C03650=1232.776,265.965,-62.554,-176.669,6.395,148.177
C03651=1232.781,265.716,-62.527,-176.671,6.393,148.177
C03652=1232.785,265.468,-62.499,-176.673,6.391,148.177
C03653=1232.790,265.219,-62.472,-176.676,6.389,148.178
C03654=1232.794,264.971,-62.445,-176.679,6.387,148.178
C03655=1232.799,264.722,-62.418,-176.681,6.385,148.178
C03656=1232.803,264.474,-62.390,-176.683,6.383,148.178
C03657=1232.807,264.225,-62.363,-176.686,6.381,148.179
C03658=1232.813,263.953,-62.332,-176.689,6.378,148.179
C03659=1232.817,263.680,-62.303,-176.691,6.376,148.179
C03660=1232.822,263.407,-62.274,-176.694,6.374,148.179
C03661=1232.827,263.135,-62.243,-176.697,6.371,148.180
C03662=1232.832,262.886,-62.216,-176.700,6.370,148.180
C03663=1232.836,262.638,-62.190,-176.702,6.367,148.180
C03664=1232.839,262.390,-62.162,-176.704,6.365,148.180
C03665=1232.844,262.141,-62.135,-176.707,6.364,148.181
C03666=1232.849,261.893,-62.108,-176.709,6.361,148.181
C03667=1232.853,261.644,-62.080,-176.712,6.359,148.181
C03668=1232.858,261.396,-62.053,-176.714,6.358,148.181
C03669=1232.863,261.147,-62.026,-176.716,6.355,148.181
C03670=1232.866,260.898,-62.000,-176.719,6.353,148.182
C03671=1232.871,260.650,-61.972,-176.721,6.352,148.182
C03672=1232.875,260.401,-61.945,-176.724,6.350,148.182
C03673=1232.880,260.153,-61.918,-176.726,6.347,148.182
C03674=1232.885,259.904,-61.891,-176.729,6.346,148.183
C03675=1232.889,259.656,-61.865,-176.731,6.344,148.183
C03676=1232.893,259.408,-61.838,-176.734,6.341,148.183
C03677=1232.898,259.159,-61.811,-176.736,6.340,148.183
C03678=1232.903,258.911,-61.784,-176.739,6.338,148.184
C03679=1232.907,258.661,-61.756,-176.741,6.335,148.184
C03680=1232.911,258.413,-61.730,-176.743,6.334,148.184
C03681=1232.915,258.165,-61.703,-176.746,6.332,148.184
C03682=1232.920,257.916,-61.676,-176.749,6.330,148.185
C03683=1232.924,257.668,-61.649,-176.751,6.328,148.185
C03684=1232.928,257.420,-61.622,-176.753,6.326,148.185
C03685=1232.933,257.171,-61.595,-176.756,6.324,148.185
C03686=1232.938,256.923,-61.568,-176.759,6.322,148.186
C03687=1232.942,256.674,-61.541,-176.761,6.320,148.186
C03688=1232.946,256.426,-61.514,-176.763,6.318,148.186
C03689=1232.951,256.177,-61.488,-176.766,6.316,148.186
C03690=1232.955,255.929,-61.462,-176.768,6.314,148.186
C03691=1232.960,255.680,-61.435,-176.771,6.312,148.187
C03692=1232.965,255.432,-61.407,-176.773,6.310,148.187
C03693=1232.968,255.183,-61.381,-176.776,6.308,148.187
C03694=1232.973,254.935,-61.354,-176.778,6.306,148.187
C03695=1232.978,254.686,-61.328,-176.781,6.304,148.188
C03696=1232.981,254.437,-61.301,-176.783,6.302,148.188
C03697=1232.986,254.188,-61.274,-176.786,6.300,148.188
C03698=1232.991,253.940,-61.247,-176.788,6.298,148.188
C03699=1232.995,253.691,-61.221,-176.791,6.296,148.189
C03700=1233.000,253.443,-61.194,-176.793,6.294,148.189
C03701=1233.004,253.194,-61.167,-176.796,6.292,148.189
C03702=1233.008,252.946,-61.140,-176.798,6.290,148.190
C03703=1233.013,252.697,-61.114,-176.800,6.288,148.190
C03704=1233.017,252.449,-61.088,-176.803,6.286,148.190
C03705=1233.022,252.200,-61.060,-176.806,6.284,148.190
C03706=1233.026,251.951,-61.035,-176.808,6.282,148.191
C03707=1233.031,251.704,-61.008,-176.810,6.280,148.191
C03708=1233.035,251.455,-60.982,-176.813,6.278,148.191
C03709=1233.040,251.206,-60.955,-176.816,6.276,148.191
C03710=1233.044,250.958,-60.929,-176.818,6.275,148.192
C03711=1233.049,250.710,-60.902,-176.821,6.273,148.192
C03712=1233.054,250.460,-60.875,-176.823,6.270,148.192
C03713=1233.058,250.212,-60.849,-176.826,6.269,148.192
C03714=1233.062,249.963,-60.823,-176.828,6.267,148.193
C03715=1233.066,249.715,-60.796,-176.831,6.265,148.193
C03716=1233.071,249.466,-60.769,-176.833,6.263,148.193
C03717=1233.075,249.218,-60.743,-176.835,6.261,148.193
C03718=1233.080,248.969,-60.716,-176.838,6.259,148.194
C03719=1233.084,248.720,-60.690,-176.841,6.257,148.194
C03720=1233.088,248.472,-60.664,-176.843,6.255,148.194
C03721=1233.093,248.223,-60.638,-176.846,6.253,148.194
C03722=1233.097,247.975,-60.611,-176.848,6.252,148.195
C03723=1233.103,247.726,-60.585,-176.850,6.250,148.195
C03724=1233.106,247.478,-60.559,-176.853,6.248,148.195
C03725=1233.111,247.229,-60.532,-176.855,6.246,148.196
C03726=1233.115,246.981,-60.506,-176.858,6.244,148.196
C03727=1233.120,246.732,-60.480,-176.860,6.242,148.196
C03728=1233.124,246.484,-60.453,-176.863,6.240,148.196
C03729=1233.128,246.235,-60.427,-176.865,6.238,148.197
C03730=1233.133,245.986,-60.401,-176.868,6.236,148.197
C03731=1233.137,245.738,-60.375,-176.871,6.234,148.197
C03732=1233.142,245.489,-60.349,-176.873,6.233,148.197
C03733=1233.147,245.241,-60.322,-176.875,6.230,148.198
C03734=1233.151,244.992,-60.296,-176.878,6.229,148.198
C03735=1233.156,244.743,-60.270,-176.880,6.227,148.198
C03736=1233.160,244.495,-60.243,-176.883,6.225,148.198
C03737=1233.164,244.246,-60.218,-176.886,6.223,148.199
C03738=1233.169,243.997,-60.191,-176.888,6.221,148.199
C03739=1233.174,243.749,-60.165,-176.890,6.220,148.199
C03740=1233.178,243.501,-60.140,-176.892,6.218,148.200
C03741=1233.183,243.252,-60.113,-176.895,6.216,148.200
C03742=1233.187,243.003,-60.087,-176.898,6.214,148.200
C03743=1233.191,242.755,-60.061,-176.900,6.212,148.200
C03744=1233.196,242.506,-60.036,-176.903,6.210,148.201
C03745=1233.201,242.257,-60.009,-176.906,6.208,148.201
C03746=1233.205,242.009,-59.983,-176.908,6.206,148.201
C03747=1233.209,241.760,-59.957,-176.910,6.204,148.201
C03748=1233.214,241.511,-59.931,-176.913,6.202,148.202
C03749=1233.219,241.263,-59.905,-176.915,6.200,148.202
C03750=1233.223,241.014,-59.880,-176.918,6.199,148.202
C03751=1233.227,240.766,-59.853,-176.921,6.197,148.203
C03752=1233.232,240.517,-59.827,-176.923,6.196,148.203
C03753=1233.236,240.268,-59.801,-176.925,6.194,148.203
C03754=1233.241,240.020,-59.776,-176.928,6.192,148.204
C03755=1233.245,239.771,-59.750,-176.930,6.190,148.204
C03756=1233.249,239.522,-59.724,-176.933,6.188,148.204
C03757=1233.254,239.274,-59.697,-176.935,6.186,148.204
C03758=1233.259,239.026,-59.672,-176.938,6.184,148.205
C03759=1233.263,238.777,-59.646,-176.941,6.182,148.205
C03760=1233.267,238.528,-59.620,-176.943,6.180,148.205
C03761=1233.271,238.279,-59.594,-176.946,6.178,148.206
C03762=1233.277,238.008,-59.567,-176.948,6.176,148.206
C03763=1233.282,237.737,-59.537,-176.951,6.175,148.206
C03764=1233.287,237.466,-59.510,-176.954,6.173,148.207
C03765=1233.292,237.194,-59.482,-176.956,6.171,148.207
C03766=1233.296,236.945,-59.456,-176.959,6.169,148.207
C03767=1233.301,236.697,-59.431,-176.961,6.167,148.208
C03768=1233.305,236.448,-59.405,-176.964,6.165,148.208
C03769=1233.309,236.199,-59.379,-176.967,6.163,148.208
C03770=1233.314,235.951,-59.354,-176.969,6.161,148.208
C03771=1233.318,235.702,-59.328,-176.971,6.159,148.209
C03772=1233.323,235.453,-59.302,-176.974,6.158,148.209
C03773=1233.327,235.205,-59.277,-176.976,6.156,148.209
C03774=1233.332,234.956,-59.250,-176.979,6.154,148.210
C03775=1233.337,234.707,-59.225,-176.981,6.153,148.210
C03776=1233.341,234.459,-59.199,-176.984,6.151,148.210
C03777=1233.346,234.210,-59.174,-176.987,6.149,148.211
C03778=1233.350,233.962,-59.148,-176.989,6.147,148.211
C03779=1233.355,233.714,-59.122,-176.992,6.145,148.211
C03780=1233.359,233.464,-59.097,-176.994,6.144,148.212
C03781=1233.363,233.215,-59.072,-176.997,6.142,148.212
C03782=1233.368,232.967,-59.046,-176.999,6.140,148.212
C03783=1233.373,232.718,-59.020,-177.002,6.138,148.213
C03784=1233.377,232.470,-58.995,-177.004,6.136,148.213
C03785=1233.382,232.221,-58.969,-177.007,6.134,148.213
C03786=1233.386,231.972,-58.944,-177.009,6.132,148.213
C03787=1233.390,231.723,-58.919,-177.012,6.130,148.214
C03788=1233.395,231.475,-58.893,-177.014,6.129,148.214
C03789=1233.399,231.226,-58.867,-177.016,6.128,148.214
C03790=1233.404,230.978,-58.842,-177.019,6.126,148.215
C03791=1233.409,230.729,-58.817,-177.022,6.124,148.215
C03792=1233.413,230.480,-58.791,-177.024,6.122,148.215
C03793=1233.418,230.232,-58.766,-177.027,6.120,148.216
C03794=1233.422,229.983,-58.740,-177.030,6.118,148.216
C03795=1233.427,229.734,-58.715,-177.032,6.117,148.216
C03796=1233.431,229.486,-58.690,-177.034,6.115,148.217
C03797=1233.435,229.237,-58.665,-177.037,6.113,148.217
C03798=1233.440,228.988,-58.640,-177.039,6.111,148.217
C03799=1233.444,228.740,-58.614,-177.042,6.110,148.218
C03800=1233.449,228.491,-58.589,-177.045,6.108,148.218
C03801=1233.454,228.242,-58.564,-177.047,6.106,148.218
C03802=1233.458,227.994,-58.538,-177.049,6.105,148.219
C03803=1233.463,227.745,-58.513,-177.052,6.103,148.219
C03804=1233.468,227.496,-58.488,-177.055,6.101,148.219
C03805=1233.471,227.248,-58.463,-177.057,6.099,148.219
C03806=1233.476,226.998,-58.438,-177.060,6.097,148.220
C03807=1233.481,226.750,-58.412,-177.062,6.095,148.220
C03808=1233.485,226.502,-58.387,-177.065,6.094,148.220
C03809=1233.490,226.253,-58.362,-177.067,6.093,148.221
C03810=1233.494,226.004,-58.336,-177.070,6.091,148.221
C03811=1233.499,225.756,-58.312,-177.072,6.089,148.221
C03812=1233.503,225.507,-58.286,-177.075,6.087,148.222
C03813=1233.508,225.258,-58.262,-177.078,6.085,148.222
C03814=1233.512,225.009,-58.236,-177.080,6.083,148.222
C03815=1233.517,224.761,-58.211,-177.082,6.082,148.223
C03816=1233.521,224.512,-58.186,-177.085,6.080,148.223
C03817=1233.526,224.263,-58.161,-177.088,6.078,148.223
C03818=1233.530,224.015,-58.136,-177.090,6.076,148.224
C03819=1233.535,223.766,-58.111,-177.093,6.075,148.224
C03820=1233.539,223.517,-58.086,-177.095,6.073,148.224
C03821=1233.544,223.269,-58.061,-177.097,6.072,148.225
C03822=1233.548,223.020,-58.035,-177.100,6.070,148.225
C03823=1233.553,222.771,-58.011,-177.103,6.068,148.225
C03824=1233.557,222.522,-57.986,-177.105,6.066,148.226
C03825=1233.562,222.274,-57.961,-177.108,6.064,148.226
C03826=1233.567,222.025,-57.936,-177.111,6.062,148.226
C03827=1233.570,221.777,-57.911,-177.113,6.061,148.227
C03828=1233.576,221.528,-57.886,-177.115,6.059,148.227
C03829=1233.580,221.278,-57.861,-177.118,6.058,148.227
C03830=1233.585,221.030,-57.836,-177.121,6.056,148.228
C03831=1233.589,220.781,-57.812,-177.123,6.054,148.228
C03832=1233.594,220.533,-57.787,-177.126,6.052,148.228
C03833=1233.598,220.284,-57.761,-177.128,6.051,148.229
C03834=1233.603,220.035,-57.737,-177.130,6.049,148.229
C03835=1233.608,219.787,-57.712,-177.133,6.047,148.229
C03836=1233.611,219.538,-57.688,-177.136,6.045,148.230
C03837=1233.616,219.289,-57.663,-177.138,6.043,148.230
C03838=1233.621,219.040,-57.638,-177.140,6.042,148.230
C03839=1233.625,218.792,-57.613,-177.143,6.041,148.231
C03840=1233.630,218.543,-57.589,-177.146,6.039,148.231
C03841=1233.635,218.294,-57.563,-177.148,6.037,148.231
C03842=1233.639,218.046,-57.539,-177.151,6.035,148.232
C03843=1233.643,217.796,-57.514,-177.154,6.033,148.232
C03844=1233.648,217.548,-57.490,-177.156,6.032,148.232
C03845=1233.653,217.299,-57.465,-177.159,6.030,148.233
C03846=1233.656,217.051,-57.440,-177.161,6.029,148.233
C03847=1233.662,216.802,-57.415,-177.164,6.027,148.234
C03848=1233.667,216.553,-57.391,-177.167,6.025,148.234
C03849=1233.671,216.304,-57.366,-177.169,6.024,148.234
C03850=1233.676,216.055,-57.342,-177.171,6.022,148.235
C03851=1233.680,215.807,-57.317,-177.174,6.020,148.235
C03852=1233.685,215.557,-57.292,-177.177,6.018,148.235
C03853=1233.689,215.310,-57.268,-177.179,6.016,148.236
C03854=1233.694,215.061,-57.243,-177.181,6.015,148.236
C03855=1233.698,214.812,-57.219,-177.184,6.013,148.236
C03856=1233.703,214.563,-57.194,-177.187,6.012,148.237
C03857=1233.707,214.315,-57.170,-177.189,6.010,148.237
C03858=1233.712,214.065,-57.145,-177.192,6.008,148.238
C03859=1233.716,213.817,-57.121,-177.194,6.007,148.238
C03860=1233.721,213.568,-57.096,-177.197,6.005,148.238
C03861=1233.725,213.319,-57.072,-177.200,6.003,148.239
C03862=1233.730,213.070,-57.047,-177.202,6.002,148.239
C03863=1233.735,212.822,-57.023,-177.204,6.000,148.239
C03864=1233.738,212.573,-56.998,-177.207,5.999,148.240
C03865=1233.743,212.324,-56.974,-177.210,5.997,148.240
C03866=1233.749,212.054,-56.947,-177.212,5.995,148.240
C03867=1233.753,211.783,-56.922,-177.215,5.993,148.241
C03868=1233.758,211.513,-56.895,-177.218,5.991,148.241
C03869=1233.763,211.242,-56.868,-177.221,5.990,148.242
C03870=1233.767,210.994,-56.844,-177.223,5.988,148.242
C03871=1233.773,210.745,-56.819,-177.226,5.986,148.242
C03872=1233.776,210.496,-56.795,-177.228,5.985,148.243
C03873=1233.782,210.247,-56.771,-177.231,5.983,148.243
C03874=1233.786,209.998,-56.747,-177.234,5.981,148.243
C03875=1233.791,209.750,-56.723,-177.236,5.980,148.244
C03876=1233.796,209.501,-56.698,-177.238,5.979,148.244
C03877=1233.799,209.252,-56.673,-177.241,5.977,148.244
C03878=1233.804,209.004,-56.649,-177.244,5.975,148.245
C03879=1233.809,208.755,-56.625,-177.246,5.973,148.245
C03880=1233.814,208.506,-56.601,-177.248,5.972,148.246
C03881=1233.817,208.257,-56.577,-177.251,5.970,148.246
C03882=1233.823,208.008,-56.552,-177.254,5.968,148.246
C03883=1233.827,207.760,-56.528,-177.257,5.967,148.247
C03884=1233.831,207.511,-56.504,-177.259,5.966,148.247
C03885=1233.837,207.262,-56.480,-177.261,5.964,148.247
C03886=1233.841,207.013,-56.456,-177.264,5.962,148.248
C03887=1233.845,206.764,-56.432,-177.267,5.960,148.248
C03888=1233.850,206.515,-56.408,-177.269,5.959,148.248
C03889=1233.855,206.267,-56.384,-177.272,5.957,148.249
C03890=1233.859,206.018,-56.360,-177.274,5.956,148.249
C03891=1233.864,205.770,-56.335,-177.277,5.954,148.250
C03892=1233.868,205.520,-56.312,-177.279,5.953,148.250
C03893=1233.873,205.271,-56.287,-177.282,5.951,148.250
C03894=1233.877,205.023,-56.263,-177.284,5.949,148.251
C03895=1233.882,204.774,-56.240,-177.287,5.947,148.251
C03896=1233.886,204.526,-56.216,-177.290,5.946,148.252
C03897=1233.892,204.277,-56.191,-177.292,5.945,148.252
C03898=1233.896,204.027,-56.167,-177.295,5.943,148.252
C03899=1233.900,203.779,-56.143,-177.297,5.942,148.253
C03900=1233.905,203.530,-56.120,-177.300,5.940,148.253
C03901=1233.909,203.281,-56.096,-177.302,5.938,148.253
C03902=1233.913,203.033,-56.072,-177.305,5.936,148.254
C03903=1233.919,202.783,-56.048,-177.307,5.935,148.254
C03904=1233.923,202.535,-56.024,-177.310,5.933,148.255
C03905=1233.928,202.286,-56.000,-177.313,5.932,148.255
C03906=1233.932,202.037,-55.976,-177.315,5.931,148.255
C03907=1233.937,201.788,-55.952,-177.317,5.929,148.256
C03908=1233.941,201.539,-55.928,-177.320,5.927,148.256
C03909=1233.946,201.290,-55.905,-177.323,5.925,148.257
C03910=1233.951,201.042,-55.880,-177.325,5.924,148.257
C03911=1233.955,200.793,-55.857,-177.328,5.922,148.257
C03912=1233.960,200.544,-55.833,-177.331,5.921,148.258
C03913=1233.965,200.295,-55.809,-177.333,5.920,148.258
C03914=1233.969,200.047,-55.785,-177.335,5.918,148.258
C03915=1233.974,199.798,-55.762,-177.338,5.916,148.259
C03916=1233.978,199.549,-55.738,-177.341,5.914,148.259
C03917=1233.983,199.300,-55.715,-177.343,5.913,148.260
C03918=1233.987,199.052,-55.691,-177.346,5.911,148.260
C03919=1233.991,198.802,-55.667,-177.348,5.910,148.260
C03920=1233.996,198.553,-55.643,-177.350,5.909,148.261
C03921=1234.000,198.305,-55.619,-177.354,5.907,148.261
C03922=1234.005,198.056,-55.596,-177.356,5.905,148.262
C03923=1234.010,197.807,-55.573,-177.358,5.904,148.262
C03924=1234.015,197.558,-55.548,-177.361,5.902,148.262
C03925=1234.020,197.309,-55.525,-177.364,5.900,148.263
C03926=1234.024,197.060,-55.501,-177.366,5.900,148.263
C03927=1234.029,196.811,-55.477,-177.369,5.898,148.264
C03928=1234.033,196.562,-55.454,-177.371,5.896,148.264
C03929=1234.038,196.313,-55.430,-177.373,5.895,148.264
C03930=1234.042,196.065,-55.407,-177.376,5.893,148.265
C03931=1234.046,195.816,-55.384,-177.379,5.891,148.265
C03932=1234.051,195.567,-55.360,-177.381,5.891,148.266
C03933=1234.055,195.319,-55.336,-177.384,5.889,148.266
C03934=1234.060,195.070,-55.313,-177.387,5.887,148.266
C03935=1234.065,194.821,-55.289,-177.389,5.886,148.267
C03936=1234.070,194.572,-55.266,-177.391,5.884,148.267
C03937=1234.074,194.323,-55.242,-177.394,5.882,148.268
C03938=1234.079,194.074,-55.219,-177.396,5.881,148.268
C03939=1234.083,193.825,-55.195,-177.399,5.880,148.268
C03940=1234.088,193.576,-55.172,-177.402,5.878,148.269
C03941=1234.093,193.327,-55.149,-177.404,5.877,148.269
C03942=1234.097,193.078,-55.125,-177.407,5.875,148.270
C03943=1234.102,192.830,-55.102,-177.410,5.873,148.270
C03944=1234.107,192.581,-55.078,-177.412,5.872,148.270
C03945=1234.111,192.333,-55.055,-177.414,5.870,148.271
C03946=1234.116,192.084,-55.032,-177.417,5.869,148.271
C03947=1234.121,191.835,-55.009,-177.420,5.868,148.272
C03948=1234.125,191.586,-54.985,-177.422,5.866,148.272
C03949=1234.130,191.337,-54.962,-177.425,5.864,148.272
C03950=1234.135,191.087,-54.939,-177.427,5.863,148.273
C03951=1234.139,190.839,-54.915,-177.430,5.862,148.273
C03952=1234.143,190.590,-54.892,-177.432,5.861,148.274
C03953=1234.148,190.341,-54.868,-177.435,5.859,148.274
C03954=1234.152,190.092,-54.845,-177.437,5.857,148.274
C03955=1234.158,189.844,-54.822,-177.440,5.856,148.275
C03956=1234.162,189.595,-54.799,-177.443,5.854,148.275
C03957=1234.166,189.346,-54.776,-177.445,5.853,148.276
C03958=1234.171,189.097,-54.753,-177.447,5.852,148.276
C03959=1234.176,188.848,-54.729,-177.450,5.850,148.276
C03960=1234.180,188.599,-54.706,-177.453,5.849,148.277
C03961=1234.185,188.350,-54.683,-177.455,5.847,148.277
C03962=1234.189,188.101,-54.660,-177.458,5.845,148.278
C03963=1234.194,187.852,-54.636,-177.460,5.844,148.278
C03964=1234.199,187.604,-54.613,-177.463,5.843,148.279
C03965=1234.204,187.355,-54.590,-177.466,5.841,148.279
C03966=1234.208,187.106,-54.567,-177.468,5.840,148.279
C03967=1234.213,186.857,-54.545,-177.470,5.838,148.280
C03968=1234.217,186.608,-54.521,-177.473,5.837,148.280
C03969=1234.221,186.359,-54.499,-177.476,5.835,148.281
C03970=1234.227,186.089,-54.473,-177.478,5.834,148.281
C03971=1234.232,185.820,-54.448,-177.481,5.832,148.282
C03972=1234.236,185.550,-54.423,-177.484,5.831,148.282
C03973=1234.242,185.281,-54.398,-177.487,5.830,148.283
C03974=1234.246,185.032,-54.375,-177.489,5.828,148.283
C03975=1234.251,184.782,-54.353,-177.491,5.827,148.283
C03976=1234.256,184.534,-54.330,-177.494,5.825,148.284
C03977=1234.261,184.285,-54.307,-177.497,5.823,148.284
C03978=1234.265,184.036,-54.284,-177.499,5.822,148.285
C03979=1234.269,183.787,-54.260,-177.502,5.820,148.285
C03980=1234.274,183.538,-54.238,-177.504,5.820,148.286
C03981=1234.279,183.290,-54.215,-177.507,5.818,148.286
C03982=1234.284,183.041,-54.192,-177.510,5.816,148.286
C03983=1234.288,182.791,-54.169,-177.512,5.815,148.287
C03984=1234.293,182.542,-54.147,-177.515,5.814,148.287
C03985=1234.298,182.294,-54.124,-177.517,5.813,148.288
C03986=1234.302,182.045,-54.101,-177.520,5.811,148.288
C03987=1234.307,181.796,-54.077,-177.522,5.809,148.288
C03988=1234.312,181.546,-54.055,-177.525,5.808,148.289
C03989=1234.315,181.298,-54.032,-177.528,5.806,148.289
C03990=1234.321,181.049,-54.009,-177.530,5.805,148.290
C03991=1234.325,180.800,-53.987,-177.533,5.804,148.290
C03992=1234.330,180.551,-53.964,-177.535,5.803,148.291
C03993=1234.334,180.303,-53.941,-177.538,5.801,148.291
C03994=1234.339,180.053,-53.919,-177.540,5.799,148.291
C03995=1234.343,179.805,-53.896,-177.543,5.798,148.292
C03996=1234.348,179.556,-53.872,-177.545,5.797,148.292
C03997=1234.353,179.307,-53.851,-177.547,5.795,148.293
C03998=1234.358,179.058,-53.827,-177.551,5.794,148.293
C03999=1234.362,178.809,-53.805,-177.553,5.793,148.294
C04000=1234.367,178.560,-53.782,-177.555,5.791,148.294
C04001=1234.371,178.311,-53.760,-177.558,5.789,148.294
C04002=1234.376,178.062,-53.737,-177.561,5.789,148.295
C04003=1234.380,177.813,-53.714,-177.563,5.787,148.295
C04004=1234.386,177.564,-53.692,-177.565,5.786,148.296
C04005=1234.390,177.315,-53.669,-177.568,5.784,148.296
C04006=1234.395,177.066,-53.647,-177.571,5.783,148.297
C04007=1234.399,176.818,-53.624,-177.573,5.781,148.297
C04008=1234.404,176.568,-53.602,-177.576,5.781,148.298
C04009=1234.408,176.319,-53.579,-177.578,5.779,148.298
C04010=1234.414,176.070,-53.556,-177.580,5.778,148.298
C04011=1234.418,175.822,-53.534,-177.584,5.776,148.299
C04012=1234.422,175.572,-53.512,-177.586,5.774,148.299
C04013=1234.427,175.324,-53.489,-177.588,5.773,148.300
C04014=1234.432,175.075,-53.467,-177.592,5.772,148.300
C04015=1234.436,174.826,-53.443,-177.594,5.771,148.301
C04016=1234.441,174.577,-53.422,-177.596,5.769,148.301
C04017=1234.445,174.328,-53.400,-177.598,5.768,148.301
C04018=1234.450,174.079,-53.376,-177.601,5.767,148.302
C04019=1234.455,173.830,-53.354,-177.604,5.766,148.302
C04020=1234.460,173.581,-53.331,-177.606,5.764,148.303
C04021=1234.465,173.332,-53.309,-177.609,5.763,148.303
C04022=1234.469,173.083,-53.287,-177.611,5.761,148.304
C04023=1234.473,172.834,-53.264,-177.614,5.760,148.304
C04024=1234.478,172.585,-53.242,-177.617,5.759,148.305
C04025=1234.483,172.336,-53.220,-177.619,5.758,148.305
C04026=1234.488,172.088,-53.197,-177.621,5.756,148.305
C04027=1234.492,171.838,-53.175,-177.624,5.755,148.306
C04028=1234.496,171.589,-53.153,-177.627,5.753,148.306
C04029=1234.502,171.341,-53.130,-177.629,5.751,148.307
C04030=1234.506,171.091,-53.108,-177.632,5.751,148.307
C04031=1234.511,170.843,-53.086,-177.635,5.749,148.308
C04032=1234.516,170.593,-53.064,-177.637,5.748,148.308
C04033=1234.520,170.345,-53.041,-177.640,5.746,148.309
C04034=1234.525,170.096,-53.019,-177.642,5.745,148.309
C04035=1234.529,169.846,-52.997,-177.645,5.744,148.310
C04036=1234.535,169.597,-52.975,-177.647,5.743,148.310
C04037=1234.539,169.349,-52.952,-177.650,5.741,148.310
C04038=1234.543,169.100,-52.931,-177.652,5.740,148.311
C04039=1234.548,168.851,-52.909,-177.655,5.739,148.311
C04040=1234.553,168.602,-52.886,-177.657,5.738,148.312
C04041=1234.558,168.352,-52.864,-177.660,5.736,148.312
C04042=1234.562,168.104,-52.842,-177.662,5.735,148.313
C04043=1234.566,167.855,-52.820,-177.665,5.733,148.313
C04044=1234.571,167.606,-52.798,-177.668,5.733,148.314
C04045=1234.576,167.357,-52.775,-177.670,5.731,148.314
C04046=1234.581,167.108,-52.754,-177.672,5.730,148.314
C04047=1234.585,166.859,-52.732,-177.675,5.728,148.315
C04048=1234.590,166.609,-52.710,-177.678,5.727,148.315
C04049=1234.594,166.361,-52.687,-177.680,5.726,148.316
C04050=1234.599,166.112,-52.665,-177.683,5.725,148.316
C04051=1234.604,165.863,-52.643,-177.685,5.724,148.317
C04052=1234.609,165.614,-52.621,-177.688,5.722,148.317
C04053=1234.613,165.365,-52.599,-177.690,5.721,148.318
C04054=1234.618,165.116,-52.578,-177.693,5.719,148.318
C04055=1234.622,164.867,-52.556,-177.695,5.719,148.319
C04056=1234.627,164.618,-52.534,-177.698,5.717,148.319
C04057=1234.632,164.369,-52.511,-177.701,5.716,148.320
C04058=1234.637,164.120,-52.490,-177.703,5.714,148.320
C04059=1234.641,163.871,-52.467,-177.705,5.713,148.320
C04060=1234.646,163.622,-52.446,-177.709,5.712,148.321
C04061=1234.651,163.373,-52.424,-177.711,5.711,148.321
C04062=1234.655,163.124,-52.402,-177.713,5.709,148.322
C04063=1234.660,162.875,-52.380,-177.716,5.708,148.322
C04064=1234.665,162.626,-52.358,-177.718,5.706,148.323
C04065=1234.669,162.377,-52.336,-177.721,5.706,148.323
C04066=1234.674,162.128,-52.315,-177.723,5.705,148.324
C04067=1234.679,161.880,-52.293,-177.726,5.703,148.324
C04068=1234.683,161.630,-52.271,-177.728,5.702,148.325
C04069=1234.688,161.382,-52.249,-177.731,5.700,148.325
C04070=1234.692,161.132,-52.228,-177.734,5.700,148.326
C04071=1234.698,160.883,-52.206,-177.736,5.698,148.326
C04072=1234.703,160.634,-52.184,-177.738,5.697,148.327
C04073=1234.707,160.385,-52.162,-177.742,5.695,148.327
C04074=1234.711,160.116,-52.138,-177.744,5.694,148.328
C04075=1234.717,159.847,-52.115,-177.747,5.693,148.328
C04076=1234.722,159.578,-52.092,-177.750,5.691,148.329
C04077=1234.727,159.309,-52.068,-177.752,5.690,148.329
C04078=1234.731,159.059,-52.047,-177.755,5.689,148.330
C04079=1234.736,158.811,-52.025,-177.757,5.688,148.330
C04080=1234.741,158.562,-52.003,-177.759,5.687,148.330
C04081=1234.745,158.313,-51.981,-177.763,5.685,148.331
C04082=1234.750,158.064,-51.960,-177.765,5.684,148.331
C04083=1234.756,157.815,-51.939,-177.768,5.683,148.332
C04084=1234.760,157.565,-51.917,-177.770,5.682,148.332
C04085=1234.765,157.317,-51.895,-177.773,5.680,148.333
C04086=1234.769,157.067,-51.873,-177.775,5.679,148.333
C04087=1234.774,156.818,-51.852,-177.778,5.678,148.334
C04088=1234.779,156.569,-51.830,-177.780,5.677,148.334
C04089=1234.783,156.320,-51.808,-177.782,5.676,148.335
C04090=1234.787,156.072,-51.787,-177.786,5.674,148.335
C04091=1234.793,155.823,-51.766,-177.788,5.673,148.336
C04092=1234.797,155.573,-51.744,-177.791,5.672,148.336
C04093=1234.802,155.325,-51.723,-177.793,5.671,148.337
C04094=1234.807,155.075,-51.702,-177.795,5.670,148.337
C04095=1234.812,154.827,-51.680,-177.798,5.668,148.338
C04096=1234.816,154.577,-51.658,-177.800,5.667,148.338
C04097=1234.821,154.328,-51.637,-177.803,5.666,148.339
C04098=1234.825,154.080,-51.616,-177.806,5.665,148.339
C04099=1234.830,153.830,-51.594,-177.808,5.664,148.340
C04100=1234.835,153.581,-51.573,-177.811,5.662,148.340
C04101=1234.840,153.332,-51.551,-177.813,5.662,148.341
C04102=1234.844,153.083,-51.530,-177.816,5.660,148.341
C04103=1234.849,152.834,-51.508,-177.818,5.659,148.342
C04104=1234.853,152.585,-51.488,-177.821,5.657,148.342
C04105=1234.858,152.336,-51.466,-177.823,5.656,148.343
C04106=1234.863,152.086,-51.445,-177.826,5.656,148.343
C04107=1234.868,151.838,-51.423,-177.829,5.654,148.344
C04108=1234.873,151.589,-51.401,-177.831,5.653,148.344
C04109=1234.877,151.340,-51.381,-177.833,5.652,148.345
C04110=1234.881,151.091,-51.359,-177.837,5.651,148.345
C04111=1234.887,150.841,-51.338,-177.839,5.650,148.346
C04112=1234.891,150.593,-51.316,-177.841,5.648,148.346
C04113=1234.896,150.344,-51.296,-177.844,5.647,148.347
C04114=1234.900,150.094,-51.275,-177.846,5.646,148.347
C04115=1234.905,149.845,-51.253,-177.849,5.645,148.348
C04116=1234.910,149.596,-51.232,-177.851,5.644,148.348
C04117=1234.915,149.348,-51.211,-177.854,5.642,148.349
C04118=1234.920,149.098,-51.190,-177.857,5.641,148.349
C04119=1234.924,148.849,-51.168,-177.859,5.641,148.350
C04120=1234.929,148.600,-51.147,-177.862,5.639,148.350
C04121=1234.933,148.352,-51.126,-177.864,5.638,148.351
C04122=1234.939,148.102,-51.105,-177.866,5.637,148.351
C04123=1234.943,147.852,-51.083,-177.870,5.636,148.352
C04124=1234.947,147.604,-51.062,-177.872,5.635,148.352
C04125=1234.952,147.355,-51.041,-177.875,5.633,148.353
C04126=1234.958,147.105,-51.020,-177.877,5.632,148.353
C04127=1234.962,146.857,-50.999,-177.880,5.632,148.354
C04128=1234.967,146.608,-50.978,-177.882,5.630,148.354
C04129=1234.971,146.358,-50.957,-177.885,5.629,148.355
C04130=1234.976,146.110,-50.936,-177.887,5.628,148.355
C04131=1234.981,145.860,-50.915,-177.890,5.626,148.355
C04132=1234.986,145.611,-50.894,-177.892,5.626,148.356
C04133=1234.990,145.363,-50.873,-177.894,5.625,148.356
C04134=1234.995,145.113,-50.852,-177.897,5.623,148.357
C04135=1234.999,144.864,-50.831,-177.900,5.622,148.357
C04136=1235.004,144.615,-50.810,-177.903,5.621,148.358
C04137=1235.009,144.366,-50.789,-177.905,5.620,148.358
C04138=1235.014,144.117,-50.768,-177.907,5.619,148.359
C04139=1235.019,143.868,-50.747,-177.910,5.617,148.359
C04140=1235.023,143.619,-50.727,-177.913,5.617,148.360
C04141=1235.028,143.370,-50.705,-177.915,5.616,148.360
C04142=1235.032,143.120,-50.684,-177.918,5.614,148.361
C04143=1235.037,142.871,-50.663,-177.920,5.613,148.361
C04144=1235.042,142.622,-50.642,-177.923,5.612,148.362
C04145=1235.047,142.373,-50.622,-177.925,5.611,148.362
C04146=1235.052,142.124,-50.600,-177.928,5.610,148.363
C04147=1235.056,141.875,-50.580,-177.930,5.609,148.363
C04148=1235.061,141.626,-50.559,-177.933,5.607,148.364
C04149=1235.066,141.377,-50.539,-177.935,5.606,148.364
C04150=1235.071,141.128,-50.518,-177.938,5.606,148.365
C04151=1235.075,140.879,-50.497,-177.941,5.604,148.366
C04152=1235.080,140.629,-50.476,-177.943,5.603,148.366
C04153=1235.084,140.381,-50.455,-177.946,5.603,148.367
C04154=1235.089,140.131,-50.434,-177.948,5.601,148.367
C04155=1235.094,139.882,-50.414,-177.951,5.600,148.368
C04156=1235.099,139.633,-50.393,-177.953,5.599,148.368
C04157=1235.103,139.384,-50.372,-177.956,5.598,148.369
C04158=1235.108,139.135,-50.351,-177.958,5.597,148.369
C04159=1235.113,138.886,-50.331,-177.961,5.596,148.370
C04160=1235.118,138.637,-50.310,-177.964,5.594,148.370
C04161=1235.122,138.388,-50.290,-177.966,5.594,148.371
C04162=1235.127,138.139,-50.269,-177.968,5.593,148.371
C04163=1235.132,137.890,-50.248,-177.971,5.592,148.372
C04164=1235.136,137.641,-50.228,-177.974,5.590,148.372
C04165=1235.142,137.391,-50.207,-177.976,5.589,148.373
C04166=1235.146,137.143,-50.187,-177.978,5.589,148.373
C04167=1235.151,136.893,-50.166,-177.982,5.587,148.374
C04168=1235.156,136.644,-50.145,-177.984,5.586,148.374
C04169=1235.160,136.395,-50.125,-177.986,5.585,148.375
C04170=1235.165,136.146,-50.104,-177.989,5.584,148.375
C04171=1235.170,135.897,-50.083,-177.992,5.583,148.376
C04172=1235.175,135.648,-50.063,-177.994,5.582,148.376
C04173=1235.179,135.399,-50.042,-177.997,5.580,148.377
C04174=1235.184,135.150,-50.022,-177.999,5.580,148.378
C04175=1235.189,134.901,-50.001,-178.001,5.579,148.378
C04176=1235.194,134.651,-49.981,-178.004,5.578,148.379
C04177=1235.198,134.402,-49.961,-178.007,5.576,148.379
C04178=1235.203,134.134,-49.938,-178.009,5.576,148.380
C04179=1235.208,133.865,-49.916,-178.013,5.574,148.380
C04180=1235.214,133.596,-49.894,-178.015,5.574,148.381
C04181=1235.218,133.328,-49.872,-178.018,5.572,148.381
C04182=1235.224,133.079,-49.851,-178.020,5.571,148.382
C04183=1235.228,132.829,-49.832,-178.023,5.570,148.382
C04184=1235.233,132.580,-49.811,-178.025,5.569,148.383
C04185=1235.237,132.331,-49.791,-178.028,5.568,148.383
C04186=1235.242,132.082,-49.770,-178.030,5.567,148.384
C04187=1235.247,131.833,-49.749,-178.033,5.566,148.385
C04188=1235.252,131.583,-49.730,-178.036,5.565,148.385
C04189=1235.257,131.334,-49.709,-178.038,5.564,148.386
C04190=1235.261,131.085,-49.688,-178.040,5.563,148.386
C04191=1235.266,130.836,-49.668,-178.043,5.562,148.387
C04192=1235.270,130.587,-49.648,-178.046,5.561,148.387
C04193=1235.276,130.337,-49.627,-178.048,5.560,148.388
C04194=1235.281,130.089,-49.607,-178.051,5.559,148.388
C04195=1235.285,129.840,-49.587,-178.053,5.558,148.389
C04196=1235.290,129.591,-49.567,-178.056,5.557,148.389
C04197=1235.294,129.342,-49.547,-178.058,5.556,148.390
C04198=1235.299,129.092,-49.526,-178.061,5.555,148.390
C04199=1235.304,128.843,-49.506,-178.064,5.554,148.391
C04200=1235.309,128.594,-49.486,-178.066,5.553,148.391
C04201=1235.313,128.345,-49.466,-178.069,5.552,148.392
C04202=1235.318,128.095,-49.446,-178.071,5.551,148.392
C04203=1235.324,127.847,-49.425,-178.074,5.550,148.393
C04204=1235.328,127.598,-49.405,-178.077,5.549,148.394
C04205=1235.333,127.348,-49.385,-178.079,5.548,148.394
C04206=1235.337,127.099,-49.365,-178.081,5.547,148.395
C04207=1235.342,126.850,-49.345,-178.084,5.545,148.395
C04208=1235.346,126.601,-49.325,-178.087,5.545,148.396
C04209=1235.351,126.352,-49.304,-178.089,5.544,148.396
C04210=1235.357,126.103,-49.285,-178.091,5.543,148.397
C04211=1235.361,125.854,-49.264,-178.094,5.542,148.397
C04212=1235.366,125.604,-49.245,-178.097,5.541,148.398
C04213=1235.370,125.355,-49.224,-178.099,5.540,148.398
C04214=1235.375,125.106,-49.205,-178.101,5.539,148.399
C04215=1235.380,124.857,-49.184,-178.104,5.538,148.399
C04216=1235.385,124.608,-49.165,-178.107,5.537,148.400
C04217=1235.389,124.359,-49.145,-178.109,5.536,148.400
C04218=1235.394,124.109,-49.125,-178.112,5.535,148.401
C04219=1235.399,123.860,-49.104,-178.114,5.534,148.401
C04220=1235.404,123.610,-49.084,-178.117,5.533,148.402
C04221=1235.409,123.362,-49.064,-178.120,5.532,148.403
C04222=1235.414,123.113,-49.045,-178.122,5.531,148.403
C04223=1235.418,122.864,-49.024,-178.124,5.531,148.404
C04224=1235.423,122.614,-49.005,-178.128,5.529,148.404
C04225=1235.427,122.365,-48.984,-178.130,5.528,148.405
C04226=1235.432,122.116,-48.965,-178.132,5.528,148.405
C04227=1235.438,121.867,-48.945,-178.134,5.527,148.406
C04228=1235.442,121.618,-48.925,-178.138,5.525,148.406
C04229=1235.447,121.368,-48.905,-178.140,5.525,148.407
C04230=1235.451,121.119,-48.885,-178.142,5.524,148.407
C04231=1235.457,120.870,-48.866,-178.145,5.523,148.408
C04232=1235.461,120.621,-48.846,-178.147,5.522,148.409
C04233=1235.466,120.372,-48.826,-178.150,5.520,148.409
C04234=1235.470,120.122,-48.806,-178.153,5.520,148.410
C04235=1235.476,119.873,-48.787,-178.155,5.519,148.410
C04236=1235.480,119.625,-48.766,-178.158,5.518,148.411
C04237=1235.485,119.375,-48.747,-178.160,5.518,148.411
C04238=1235.490,119.125,-48.727,-178.163,5.516,148.412
C04239=1235.495,118.877,-48.707,-178.165,5.515,148.413
C04240=1235.499,118.628,-48.687,-178.168,5.514,148.413
C04241=1235.504,118.378,-48.668,-178.170,5.514,148.414
C04242=1235.509,118.130,-48.648,-178.173,5.513,148.414
C04243=1235.514,117.880,-48.628,-178.175,5.511,148.415
C04244=1235.518,117.631,-48.609,-178.178,5.510,148.415
C04245=1235.523,117.381,-48.589,-178.181,5.510,148.416
C04246=1235.528,117.133,-48.569,-178.183,5.509,148.416
C04247=1235.533,116.884,-48.550,-178.185,5.508,148.417
C04248=1235.537,116.634,-48.530,-178.189,5.507,148.418
C04249=1235.543,116.385,-48.511,-178.191,5.506,148.418
C04250=1235.547,116.136,-48.490,-178.193,5.505,148.419
C04251=1235.552,115.887,-48.471,-178.196,5.504,148.419
C04252=1235.557,115.638,-48.451,-178.198,5.504,148.420
C04253=1235.561,115.388,-48.432,-178.201,5.502,148.420
C04254=1235.566,115.139,-48.413,-178.204,5.501,148.421
C04255=1235.571,114.891,-48.393,-178.206,5.500,148.421
C04256=1235.576,114.641,-48.373,-178.209,5.500,148.422
C04257=1235.580,114.392,-48.353,-178.211,5.499,148.422
C04258=1235.586,114.143,-48.334,-178.214,5.497,148.423
C04259=1235.591,113.893,-48.314,-178.216,5.497,148.424
C04260=1235.595,113.644,-48.295,-178.219,5.496,148.424
C04261=1235.600,113.395,-48.276,-178.221,5.495,148.425
C04262=1235.605,113.145,-48.256,-178.224,5.494,148.425
C04263=1235.609,112.896,-48.237,-178.226,5.494,148.426
C04264=1235.614,112.648,-48.217,-178.229,5.492,148.426
C04265=1235.618,112.398,-48.198,-178.232,5.491,148.427
C04266=1235.623,112.149,-48.178,-178.234,5.490,148.427
C04267=1235.628,111.900,-48.159,-178.236,5.490,148.428
C04268=1235.633,111.650,-48.139,-178.239,5.489,148.429
C04269=1235.639,111.401,-48.120,-178.241,5.488,148.429
C04270=1235.643,111.152,-48.101,-178.244,5.487,148.430
C04271=1235.647,110.903,-48.081,-178.247,5.486,148.430
C04272=1235.653,110.654,-48.062,-178.249,5.485,148.431
C04273=1235.657,110.404,-48.042,-178.252,5.485,148.431
C04274=1235.662,110.156,-48.023,-178.254,5.484,148.432
C04275=1235.667,109.906,-48.004,-178.256,5.483,148.433
C04276=1235.671,109.656,-47.984,-178.260,5.481,148.433
C04277=1235.676,109.408,-47.965,-178.262,5.481,148.434
C04278=1235.681,109.158,-47.946,-178.265,5.480,148.434
C04279=1235.686,108.909,-47.926,-178.267,5.479,148.435
C04280=1235.691,108.660,-47.907,-178.270,5.479,148.435
C04281=1235.696,108.411,-47.888,-178.272,5.478,148.436
C04282=1235.701,108.142,-47.868,-178.275,5.476,148.437
C04283=1235.706,107.873,-47.847,-178.277,5.476,148.437
C04284=1235.711,107.606,-47.826,-178.280,5.475,148.438
C04285=1235.716,107.337,-47.805,-178.283,5.473,148.438
C04286=1235.721,107.088,-47.786,-178.286,5.473,148.439
C04287=1235.725,106.839,-47.766,-178.288,5.472,148.440
C04288=1235.731,106.589,-47.748,-178.291,5.471,148.440
C04289=1235.735,106.340,-47.729,-178.293,5.471,148.441
C04290=1235.740,106.091,-47.710,-178.296,5.470,148.441
C04291=1235.745,105.842,-47.690,-178.298,5.469,148.442
C04292=1235.749,105.592,-47.671,-178.301,5.468,148.442
C04293=1235.755,105.343,-47.652,-178.304,5.467,148.443
C04294=1235.760,105.093,-47.633,-178.306,5.466,148.444
C04295=1235.764,104.845,-47.614,-178.308,5.465,148.444
C04296=1235.769,104.595,-47.594,-178.311,5.465,148.445
C04297=1235.774,104.347,-47.576,-178.314,5.464,148.445
C04298=1235.778,104.097,-47.556,-178.316,5.463,148.446
C04299=1235.784,103.847,-47.537,-178.318,5.463,148.447
C04300=1235.788,103.598,-47.518,-178.322,5.461,148.447
C04301=1235.793,103.349,-47.499,-178.324,5.460,148.448
C04302=1235.797,103.100,-47.480,-178.326,5.459,148.448
C04303=1235.803,102.851,-47.461,-178.329,5.459,148.449
C04304=1235.808,102.602,-47.443,-178.331,5.458,148.449
C04305=1235.812,102.353,-47.423,-178.334,5.457,148.450
C04306=1235.817,102.103,-47.405,-178.336,5.457,148.451
C04307=1235.822,101.854,-47.385,-178.339,5.456,148.451
C04308=1235.827,101.605,-47.366,-178.341,5.455,148.452
C04309=1235.831,101.356,-47.347,-178.344,5.454,148.452
C04310=1235.837,101.106,-47.328,-178.347,5.453,148.453
C04311=1235.841,100.857,-47.309,-178.349,5.452,148.454
C04312=1235.846,100.608,-47.290,-178.352,5.451,148.454
C04313=1235.851,100.358,-47.272,-178.354,5.451,148.455
C04314=1235.856,100.109,-47.252,-178.357,5.450,148.455
C04315=1235.861,99.860,-47.234,-178.359,5.449,148.456
C04316=1235.865,99.611,-47.215,-178.362,5.449,148.456
C04317=1235.870,99.362,-47.196,-178.364,5.448,148.457
C04318=1235.875,99.112,-47.178,-178.367,5.447,148.458
C04319=1235.880,98.863,-47.158,-178.369,5.446,148.458
C04320=1235.884,98.613,-47.140,-178.372,5.445,148.459
C04321=1235.890,98.364,-47.121,-178.375,5.444,148.459
C04322=1235.894,98.116,-47.102,-178.377,5.444,148.460
C04323=1235.899,97.866,-47.083,-178.379,5.443,148.460
C04324=1235.904,97.617,-47.065,-178.382,5.442,148.461
C04325=1235.908,97.367,-47.046,-178.385,5.441,148.462
C04326=1235.913,97.118,-47.027,-178.387,5.441,148.462
C04327=1235.918,96.869,-47.009,-178.389,5.440,148.463
C04328=1235.923,96.620,-46.989,-178.392,5.439,148.463
C04329=1235.928,96.371,-46.971,-178.395,5.438,148.464
C04330=1235.933,96.122,-46.952,-178.397,5.437,148.465
C04331=1235.938,95.872,-46.934,-178.400,5.436,148.465
C04332=1235.942,95.623,-46.915,-178.403,5.436,148.466
C04333=1235.947,95.373,-46.896,-178.405,5.435,148.466
C04334=1235.952,95.124,-46.877,-178.407,5.434,148.467
C04335=1235.957,94.875,-46.859,-178.410,5.433,148.468
C04336=1235.962,94.626,-46.840,-178.413,5.433,148.468
C04337=1235.966,94.377,-46.822,-178.415,5.432,148.469
C04338=1235.971,94.127,-46.804,-178.417,5.431,148.469
C04339=1235.976,93.878,-46.784,-178.420,5.431,148.470
C04340=1235.981,93.629,-46.766,-178.423,5.430,148.471
C04341=1235.986,93.380,-46.747,-178.426,5.429,148.471
C04342=1235.991,93.130,-46.728,-178.428,5.428,148.472
C04343=1235.996,92.881,-46.710,-178.431,5.427,148.472
C04344=1236.000,92.632,-46.692,-178.433,5.426,148.473
C04345=1236.005,92.382,-46.673,-178.436,5.426,148.474
C04346=1236.010,92.133,-46.654,-178.438,5.425,148.474
C04347=1236.015,91.884,-46.636,-178.440,5.424,148.475
C04348=1236.020,91.634,-46.617,-178.443,5.424,148.475
C04349=1236.024,91.386,-46.598,-178.446,5.423,148.476
C04350=1236.029,91.136,-46.581,-178.448,5.422,148.477
C04351=1236.034,90.887,-46.563,-178.450,5.421,148.477
C04352=1236.039,90.638,-46.543,-178.453,5.421,148.478
C04353=1236.044,90.388,-46.525,-178.456,5.420,148.478
C04354=1236.049,90.139,-46.507,-178.458,5.420,148.479
C04355=1236.053,89.889,-46.489,-178.460,5.419,148.479
C04356=1236.058,89.640,-46.469,-178.463,5.418,148.480
C04357=1236.063,89.391,-46.451,-178.466,5.417,148.481
C04358=1236.068,89.142,-46.433,-178.469,5.416,148.481
C04359=1236.073,88.892,-46.415,-178.472,5.415,148.482
C04360=1236.077,88.644,-46.396,-178.474,5.414,148.482
C04361=1236.083,88.394,-46.378,-178.476,5.414,148.483
C04362=1236.088,88.145,-46.360,-178.479,5.413,148.484
C04363=1236.092,87.895,-46.341,-178.482,5.413,148.484
C04364=1236.097,87.647,-46.323,-178.484,5.412,148.485
C04365=1236.102,87.397,-46.305,-178.486,5.411,148.485
C04366=1236.107,87.148,-46.286,-178.489,5.410,148.486
C04367=1236.112,86.898,-46.268,-178.492,5.410,148.487
C04368=1236.116,86.649,-46.250,-178.494,5.409,148.487
C04369=1236.121,86.400,-46.232,-178.496,5.408,148.488
C04370=1236.126,86.151,-46.213,-178.499,5.408,148.489
C04371=1236.130,85.901,-46.195,-178.502,5.407,148.489
C04372=1236.136,85.652,-46.176,-178.504,5.406,148.490
C04373=1236.141,85.403,-46.158,-178.507,5.406,148.490
C04374=1236.146,85.153,-46.140,-178.509,5.405,148.491
C04375=1236.151,84.904,-46.122,-178.512,5.404,148.492
C04376=1236.155,84.654,-46.104,-178.514,5.404,148.492
C04377=1236.160,84.405,-46.086,-178.517,5.403,148.493
C04378=1236.165,84.156,-46.068,-178.519,5.402,148.493
C04379=1236.169,83.907,-46.049,-178.522,5.401,148.494
C04380=1236.174,83.658,-46.031,-178.524,5.401,148.495
C04381=1236.179,83.408,-46.013,-178.527,5.400,148.495
C04382=1236.184,83.159,-45.994,-178.529,5.400,148.496
C04383=1236.189,82.910,-45.976,-178.532,5.399,148.496
C04384=1236.194,82.661,-45.958,-178.534,5.398,148.497
C04385=1236.199,82.411,-45.940,-178.537,5.397,148.498
C04386=1236.204,82.143,-45.921,-178.540,5.396,148.498
C04387=1236.209,81.875,-45.902,-178.543,5.395,148.499
C04388=1236.215,81.606,-45.883,-178.545,5.395,148.500
C04389=1236.220,81.338,-45.864,-178.548,5.394,148.500
C04390=1236.225,81.089,-45.846,-178.550,5.394,148.501
C04391=1236.229,80.839,-45.827,-178.553,5.393,148.502
C04392=1236.235,80.589,-45.809,-178.556,5.392,148.502
C04393=1236.239,80.340,-45.791,-178.558,5.391,148.503
C04394=1236.244,80.091,-45.773,-178.560,5.391,148.503
C04395=1236.249,79.842,-45.755,-178.563,5.390,148.504
C04396=1236.254,79.593,-45.737,-178.566,5.390,148.505
C04397=1236.259,79.343,-45.719,-178.568,5.389,148.505
C04398=1236.264,79.094,-45.701,-178.571,5.388,148.506
C04399=1236.268,78.845,-45.683,-178.573,5.387,148.506
C04400=1236.273,78.595,-45.665,-178.576,5.387,148.507
C04401=1236.278,78.346,-45.648,-178.578,5.386,148.508
C04402=1236.283,78.096,-45.630,-178.581,5.386,148.508
C04403=1236.288,77.847,-45.612,-178.584,5.385,148.509
C04404=1236.292,77.598,-45.594,-178.586,5.384,148.509
C04405=1236.297,77.349,-45.576,-178.588,5.383,148.510
C04406=1236.302,77.100,-45.558,-178.591,5.383,148.511
C04407=1236.307,76.851,-45.540,-178.594,5.382,148.511
C04408=1236.312,76.601,-45.523,-178.596,5.382,148.512
C04409=1236.317,76.352,-45.505,-178.599,5.381,148.513
C04410=1236.322,76.102,-45.486,-178.601,5.380,148.513
C04411=1236.327,75.853,-45.468,-178.604,5.380,148.514
C04412=1236.331,75.603,-45.450,-178.606,5.379,148.514
C04413=1236.337,75.354,-45.433,-178.609,5.378,148.515
C04414=1236.341,75.105,-45.416,-178.612,5.378,148.516
C04415=1236.346,74.856,-45.398,-178.614,5.377,148.516
C04416=1236.351,74.606,-45.380,-178.616,5.376,148.517
C04417=1236.356,74.357,-45.362,-178.619,5.376,148.518
C04418=1236.361,74.107,-45.344,-178.622,5.375,148.518
C04419=1236.366,73.858,-45.326,-178.624,5.374,148.519
C04420=1236.371,73.609,-45.308,-178.627,5.374,148.520
C04421=1236.375,73.360,-45.292,-178.629,5.373,148.520
C04422=1236.380,73.110,-45.274,-178.632,5.372,148.521
C04423=1236.385,72.861,-45.256,-178.634,5.372,148.521
C04424=1236.390,72.611,-45.239,-178.637,5.371,148.522
C04425=1236.395,72.362,-45.221,-178.639,5.370,148.523
C04426=1236.400,72.113,-45.203,-178.642,5.370,148.523
C04427=1236.404,71.864,-45.186,-178.645,5.369,148.524
C04428=1236.409,71.614,-45.168,-178.647,5.369,148.525
C04429=1236.414,71.365,-45.150,-178.649,5.368,148.525
C04430=1236.420,71.115,-45.133,-178.652,5.367,148.526
C04431=1236.424,70.866,-45.115,-178.655,5.366,148.526
C04432=1236.429,70.617,-45.097,-178.657,5.366,148.527
C04433=1236.434,70.368,-45.080,-178.659,5.366,148.528
C04434=1236.439,70.118,-45.062,-178.662,5.366,148.528
C04435=1236.444,69.869,-45.045,-178.665,5.365,148.529
C04436=1236.448,69.620,-45.027,-178.667,5.364,148.529
C04437=1236.453,69.371,-45.010,-178.669,5.363,148.530
C04438=1236.458,69.121,-44.992,-178.672,5.363,148.531
C04439=1236.463,68.872,-44.974,-178.675,5.362,148.531
C04440=1236.468,68.622,-44.958,-178.677,5.362,148.532
C04441=1236.473,68.373,-44.940,-178.680,5.361,148.533
C04442=1236.478,68.123,-44.922,-178.683,5.360,148.533
C04443=1236.483,67.874,-44.904,-178.685,5.359,148.534
C04444=1236.487,67.625,-44.888,-178.687,5.359,148.534
C04445=1236.492,67.375,-44.870,-178.690,5.358,148.535
C04446=1236.497,67.126,-44.852,-178.693,5.358,148.536
C04447=1236.502,66.877,-44.835,-178.695,5.357,148.536
C04448=1236.507,66.628,-44.818,-178.698,5.356,148.537
C04449=1236.512,66.378,-44.800,-178.700,5.356,148.538
C04450=1236.517,66.129,-44.784,-178.703,5.355,148.538
C04451=1236.522,65.880,-44.766,-178.705,5.354,148.539
C04452=1236.527,65.630,-44.748,-178.707,5.355,148.540
C04453=1236.531,65.381,-44.731,-178.710,5.354,148.540
C04454=1236.536,65.131,-44.714,-178.713,5.353,148.541
C04455=1236.541,64.882,-44.696,-178.715,5.353,148.542
C04456=1236.546,64.633,-44.679,-178.718,5.352,148.542
C04457=1236.551,64.383,-44.662,-178.720,5.352,148.543
C04458=1236.556,64.134,-44.644,-178.723,5.351,148.544
C04459=1236.561,63.885,-44.627,-178.725,5.350,148.544
C04460=1236.566,63.635,-44.610,-178.728,5.350,148.545
C04461=1236.570,63.386,-44.593,-178.731,5.349,148.545
C04462=1236.575,63.136,-44.576,-178.733,5.348,148.546
C04463=1236.580,62.887,-44.558,-178.736,5.348,148.547
C04464=1236.585,62.638,-44.541,-178.738,5.347,148.547
C04465=1236.590,62.388,-44.524,-178.741,5.347,148.548
C04466=1236.595,62.140,-44.507,-178.744,5.346,148.549
C04467=1236.600,61.890,-44.489,-178.745,5.346,148.549
C04468=1236.605,61.640,-44.472,-178.748,5.345,148.550
C04469=1236.609,61.391,-44.455,-178.750,5.345,148.550
C04470=1236.615,61.142,-44.437,-178.753,5.344,148.551
C04471=1236.619,60.892,-44.421,-178.756,5.343,148.552
C04472=1236.625,60.643,-44.404,-178.758,5.343,148.552
C04473=1236.629,60.394,-44.386,-178.761,5.342,148.553
C04474=1236.634,60.144,-44.369,-178.764,5.342,148.554
C04475=1236.639,59.895,-44.353,-178.766,5.341,148.554
C04476=1236.644,59.645,-44.335,-178.769,5.341,148.555
C04477=1236.648,59.396,-44.318,-178.771,5.340,148.555
C04478=1236.654,59.147,-44.301,-178.773,5.340,148.556
C04479=1236.659,58.897,-44.284,-178.776,5.339,148.557
C04480=1236.664,58.648,-44.267,-178.778,5.339,148.558
C04481=1236.669,58.399,-44.249,-178.781,5.338,148.558
C04482=1236.673,58.149,-44.232,-178.784,5.338,148.559
C04483=1236.678,57.900,-44.216,-178.786,5.337,148.560
C04484=1236.683,57.651,-44.199,-178.789,5.336,148.560
C04485=1236.688,57.401,-44.182,-178.792,5.336,148.561
C04486=1236.693,57.152,-44.164,-178.794,5.335,148.562
C04487=1236.697,56.902,-44.148,-178.796,5.334,148.562
C04488=1236.703,56.653,-44.131,-178.799,5.334,148.563
C04489=1236.708,56.404,-44.114,-178.801,5.334,148.563
C04490=1236.713,56.135,-44.095,-178.804,5.333,148.564
C04491=1236.718,55.867,-44.078,-178.806,5.333,148.565
C04492=1236.724,55.598,-44.059,-178.810,5.332,148.566
C04493=1236.729,55.330,-44.041,-178.813,5.331,148.566
C04494=1236.734,55.081,-44.024,-178.815,5.331,148.567
C04495=1236.739,54.831,-44.007,-178.817,5.331,148.568
C04496=1236.744,54.581,-43.990,-178.820,5.330,148.568
C04497=1236.749,54.333,-43.974,-178.822,5.329,148.569
C04498=1236.753,54.083,-43.957,-178.825,5.329,148.569
C04499=1236.759,53.833,-43.940,-178.827,5.328,148.570
C04500=1236.763,53.584,-43.923,-178.830,5.327,148.571
C04501=1236.769,53.335,-43.906,-178.833,5.327,148.571
C04502=1236.773,53.085,-43.889,-178.835,5.326,148.572
C04503=1236.777,52.836,-43.872,-178.837,5.327,148.573
C04504=1236.783,52.587,-43.855,-178.840,5.326,148.573
C04505=1236.788,52.338,-43.838,-178.843,5.325,148.574
C04506=1236.792,52.088,-43.822,-178.845,5.325,148.575
C04507=1236.797,51.838,-43.805,-178.848,5.324,148.575
C04508=1236.803,51.590,-43.788,-178.851,5.324,148.576
C04509=1236.807,51.340,-43.772,-178.853,5.323,148.576
C04510=1236.813,51.090,-43.755,-178.855,5.322,148.577
C04511=1236.818,50.841,-43.739,-178.857,5.322,148.578
C04512=1236.822,50.592,-43.722,-178.860,5.322,148.578
C04513=1236.827,50.342,-43.705,-178.863,5.321,148.579
C04514=1236.832,50.093,-43.688,-178.865,5.321,148.580
C04515=1236.837,49.843,-43.672,-178.868,5.320,148.580
C04516=1236.841,49.594,-43.655,-178.871,5.319,148.581
C04517=1236.847,49.345,-43.638,-178.873,5.319,148.582
C04518=1236.852,49.095,-43.622,-178.876,5.318,148.582
C04519=1236.856,48.846,-43.605,-178.878,5.319,148.583
C04520=1236.862,48.597,-43.588,-178.881,5.318,148.584
C04521=1236.866,48.347,-43.571,-178.883,5.317,148.584
C04522=1236.871,48.097,-43.555,-178.886,5.317,148.585
C04523=1236.876,47.848,-43.539,-178.888,5.316,148.586
C04524=1236.882,47.599,-43.522,-178.891,5.315,148.586
C04525=1236.886,47.349,-43.505,-178.893,5.315,148.587
C04526=1236.891,47.100,-43.489,-178.895,5.315,148.588
C04527=1236.896,46.851,-43.472,-178.898,5.314,148.588
C04528=1236.901,46.600,-43.456,-178.901,5.314,148.589
C04529=1236.906,46.352,-43.439,-178.903,5.313,148.590
C04530=1236.911,46.102,-43.423,-178.906,5.313,148.590
C04531=1236.916,45.853,-43.406,-178.909,5.312,148.591
C04532=1236.920,45.604,-43.390,-178.911,5.312,148.592
C04533=1236.926,45.354,-43.373,-178.913,5.312,148.592
C04534=1236.931,45.105,-43.357,-178.916,5.311,148.593
C04535=1236.935,44.855,-43.340,-178.918,5.311,148.594
C04536=1236.940,44.606,-43.324,-178.921,5.310,148.594
C04537=1236.945,44.357,-43.307,-178.924,5.309,148.595
C04538=1236.950,44.107,-43.291,-178.926,5.309,148.596
C04539=1236.955,43.858,-43.274,-178.928,5.309,148.596
C04540=1236.960,43.608,-43.258,-178.931,5.309,148.597
C04541=1236.965,43.359,-43.242,-178.933,5.308,148.597
C04542=1236.970,43.109,-43.225,-178.936,5.307,148.598
C04543=1236.975,42.861,-43.209,-178.939,5.306,148.599
C04544=1236.979,42.611,-43.192,-178.941,5.306,148.599
C04545=1236.985,42.361,-43.176,-178.943,5.306,148.600
C04546=1236.990,42.112,-43.160,-178.946,5.306,148.601
C04547=1236.994,41.862,-43.143,-178.949,5.305,148.602
C04548=1237.000,41.613,-43.127,-178.951,5.304,148.602
C04549=1237.004,41.364,-43.111,-178.954,5.304,148.603
C04550=1237.010,41.114,-43.095,-178.956,5.303,148.604
C04551=1237.014,40.865,-43.078,-178.959,5.304,148.604
C04552=1237.019,40.616,-43.062,-178.961,5.303,148.605
C04553=1237.024,40.366,-43.046,-178.964,5.302,148.606
C04554=1237.029,40.117,-43.030,-178.966,5.302,148.606
C04555=1237.034,39.867,-43.013,-178.969,5.301,148.607
C04556=1237.039,39.617,-42.997,-178.972,5.301,148.608
C04557=1237.044,39.368,-42.980,-178.974,5.301,148.608
C04558=1237.049,39.118,-42.964,-178.976,5.300,148.609
C04559=1237.054,38.869,-42.948,-178.979,5.300,148.610
C04560=1237.059,38.619,-42.932,-178.982,5.299,148.610
C04561=1237.064,38.371,-42.916,-178.984,5.299,148.611
C04562=1237.068,38.121,-42.899,-178.987,5.298,148.612
C04563=1237.074,37.872,-42.884,-178.989,5.298,148.612
C04564=1237.078,37.622,-42.867,-178.992,5.298,148.613
C04565=1237.084,37.373,-42.851,-178.994,5.297,148.614
C04566=1237.088,37.123,-42.835,-178.997,5.297,148.614
C04567=1237.094,36.874,-42.819,-178.999,5.296,148.615
C04568=1237.099,36.625,-42.803,-179.001,5.296,148.615
C04569=1237.103,36.375,-42.787,-179.004,5.295,148.616
C04570=1237.109,36.126,-42.770,-179.006,5.295,148.617
C04571=1237.113,35.876,-42.755,-179.009,5.294,148.618
C04572=1237.118,35.627,-42.738,-179.012,5.294,148.618
C04573=1237.123,35.377,-42.722,-179.014,5.293,148.619
C04574=1237.129,35.128,-42.707,-179.016,5.293,148.620
C04575=1237.133,34.878,-42.690,-179.019,5.293,148.620
C04576=1237.138,34.629,-42.674,-179.022,5.292,148.621
C04577=1237.143,34.379,-42.658,-179.024,5.292,148.622
C04578=1237.148,34.130,-42.642,-179.027,5.291,148.622
C04579=1237.153,33.881,-42.625,-179.029,5.291,148.623
C04580=1237.158,33.631,-42.610,-179.032,5.291,148.624
C04581=1237.163,33.382,-42.595,-179.034,5.290,148.624
C04582=1237.167,33.133,-42.578,-179.037,5.290,148.625
C04583=1237.173,32.883,-42.563,-179.040,5.289,148.626
C04584=1237.177,32.634,-42.546,-179.042,5.289,148.626
C04585=1237.183,32.384,-42.530,-179.044,5.289,148.627
C04586=1237.187,32.134,-42.514,-179.047,5.288,148.628
C04587=1237.192,31.885,-42.498,-179.050,5.288,148.628
C04588=1237.198,31.636,-42.483,-179.052,5.287,148.629
C04589=1237.203,31.386,-42.467,-179.054,5.287,148.630
C04590=1237.208,31.137,-42.450,-179.057,5.287,148.630
C04591=1237.212,30.887,-42.435,-179.060,5.286,148.631
C04592=1237.217,30.638,-42.419,-179.062,5.286,148.632
C04593=1237.223,30.389,-42.404,-179.064,5.286,148.632
C04594=1237.227,30.119,-42.386,-179.067,5.285,148.633
C04595=1237.233,29.852,-42.369,-179.070,5.285,148.634
C04596=1237.238,29.583,-42.352,-179.073,5.285,148.635
C04597=1237.244,29.315,-42.335,-179.075,5.284,148.635
C04598=1237.249,29.064,-42.319,-179.078,5.283,148.636
C04599=1237.253,28.815,-42.304,-179.081,5.283,148.637
C04600=1237.259,28.566,-42.288,-179.083,5.282,148.637
C04601=1237.263,28.316,-42.271,-179.085,5.283,148.638
C04602=1237.269,28.067,-42.256,-179.088,5.282,148.639
C04603=1237.274,27.818,-42.240,-179.091,5.282,148.639
C04604=1237.278,27.568,-42.225,-179.093,5.281,148.640
C04605=1237.283,27.318,-42.209,-179.096,5.281,148.641
C04606=1237.288,27.070,-42.193,-179.098,5.281,148.641
C04607=1237.293,26.820,-42.177,-179.101,5.280,148.642
C04608=1237.299,26.570,-42.161,-179.103,5.280,148.643
C04609=1237.303,26.321,-42.146,-179.106,5.279,148.644
C04610=1237.308,26.071,-42.130,-179.108,5.279,148.644
C04611=1237.313,25.822,-42.115,-179.111,5.279,148.645
C04612=1237.318,25.573,-42.099,-179.113,5.278,148.646
C04613=1237.323,25.323,-42.083,-179.116,5.278,148.646
C04614=1237.328,25.074,-42.068,-179.118,5.278,148.647
C04615=1237.333,24.824,-42.052,-179.121,5.277,148.648
C04616=1237.338,24.574,-42.036,-179.123,5.277,148.648
C04617=1237.343,24.325,-42.021,-179.126,5.276,148.649
C04618=1237.348,24.076,-42.006,-179.128,5.276,148.650
C04619=1237.354,23.826,-41.990,-179.131,5.276,148.650
C04620=1237.358,23.576,-41.975,-179.133,5.275,148.651
C04621=1237.363,23.327,-41.959,-179.136,5.275,148.652
C04622=1237.368,23.078,-41.943,-179.139,5.274,148.652
C04623=1237.372,22.828,-41.927,-179.141,5.274,148.653
C04624=1237.377,22.579,-41.912,-179.143,5.274,148.654
C04625=1237.383,22.330,-41.896,-179.146,5.273,148.654
C04626=1237.388,22.081,-41.881,-179.149,5.273,148.655
C04627=1237.392,21.830,-41.865,-179.151,5.273,148.656
C04628=1237.398,21.581,-41.850,-179.153,5.272,148.656
C04629=1237.402,21.332,-41.835,-179.156,5.272,148.657
C04630=1237.408,21.083,-41.819,-179.159,5.271,148.658
C04631=1237.413,20.832,-41.803,-179.161,5.272,148.659
C04632=1237.417,20.583,-41.788,-179.164,5.271,148.659
C04633=1237.423,20.334,-41.773,-179.166,5.271,148.660
C04634=1237.428,20.085,-41.757,-179.169,5.270,148.661
C04635=1237.432,19.835,-41.742,-179.171,5.270,148.661
C04636=1237.437,19.585,-41.726,-179.174,5.270,148.662
C04637=1237.443,19.336,-41.710,-179.176,5.269,148.663
C04638=1237.447,19.087,-41.695,-179.179,5.269,148.663
C04639=1237.452,18.836,-41.680,-179.181,5.269,148.664
C04640=1237.457,18.587,-41.665,-179.184,5.268,148.665
C04641=1237.463,18.338,-41.650,-179.186,5.268,148.665
C04642=1237.468,18.088,-41.634,-179.189,5.267,148.666
C04643=1237.473,17.839,-41.619,-179.191,5.267,148.667
C04644=1237.477,17.589,-41.603,-179.194,5.267,148.667
C04645=1237.482,17.340,-41.588,-179.196,5.266,148.668
C04646=1237.487,17.091,-41.572,-179.199,5.266,148.669
C04647=1237.492,16.841,-41.557,-179.201,5.266,148.669
C04648=1237.498,16.591,-41.543,-179.204,5.266,148.670
C04649=1237.502,16.342,-41.527,-179.206,5.265,148.671
C04650=1237.507,16.092,-41.512,-179.208,5.265,148.672
C04651=1237.513,15.843,-41.496,-179.211,5.265,148.672
C04652=1237.517,15.594,-41.481,-179.214,5.264,148.673
C04653=1237.523,15.344,-41.465,-179.216,5.264,148.674
C04654=1237.528,15.095,-41.451,-179.218,5.264,148.674
C04655=1237.532,14.845,-41.435,-179.221,5.263,148.675
C04656=1237.537,14.595,-41.420,-179.224,5.263,148.676
C04657=1237.542,14.346,-41.405,-179.226,5.262,148.676
C04658=1237.547,14.097,-41.390,-179.229,5.263,148.677
C04659=1237.553,13.847,-41.375,-179.231,5.262,148.678
C04660=1237.557,13.598,-41.360,-179.234,5.262,148.679
C04661=1237.562,13.348,-41.344,-179.237,5.261,148.679
C04662=1237.567,13.099,-41.329,-179.239,5.261,148.680
C04663=1237.572,12.849,-41.314,-179.242,5.261,148.681
C04664=1237.577,12.600,-41.299,-179.244,5.260,148.681
C04665=1237.582,12.350,-41.284,-179.246,5.261,148.682
C04666=1237.587,12.101,-41.268,-179.249,5.260,148.683
C04667=1237.592,11.851,-41.254,-179.252,5.260,148.683
C04668=1237.597,11.602,-41.239,-179.254,5.259,148.684
C04669=1237.602,11.352,-41.223,-179.256,5.259,148.685
C04670=1237.607,11.102,-41.208,-179.259,5.259,148.685
C04671=1237.612,10.853,-41.193,-179.262,5.258,148.686
C04672=1237.617,10.604,-41.178,-179.264,5.258,148.687
C04673=1237.622,10.354,-41.163,-179.266,5.258,148.687
C04674=1237.627,10.105,-41.148,-179.269,5.257,148.688
C04675=1237.632,9.855,-41.133,-179.272,5.257,148.689
C04676=1237.637,9.606,-41.119,-179.274,5.257,148.690
C04677=1237.643,9.356,-41.103,-179.276,5.257,148.690
C04678=1237.647,9.107,-41.088,-179.279,5.256,148.691
C04679=1237.652,8.857,-41.073,-179.281,5.256,148.692
C04680=1237.657,8.607,-41.058,-179.284,5.256,148.692
C04681=1237.662,8.358,-41.043,-179.286,5.255,148.693
C04682=1237.667,8.109,-41.029,-179.289,5.255,148.694
C04683=1237.672,7.859,-41.013,-179.291,5.255,148.694
C04684=1237.677,7.609,-40.999,-179.294,5.254,148.695
C04685=1237.682,7.360,-40.984,-179.296,5.254,148.696
C04686=1237.687,7.110,-40.969,-179.299,5.254,148.697
C04687=1237.692,6.861,-40.954,-179.302,5.254,148.697
C04688=1237.697,6.612,-40.939,-179.304,5.253,148.698
C04689=1237.702,6.362,-40.924,-179.306,5.254,148.699
C04690=1237.707,6.113,-40.909,-179.309,5.253,148.699
C04691=1237.712,5.863,-40.895,-179.312,5.253,148.700
C04692=1237.717,5.614,-40.879,-179.314,5.252,148.701
C04693=1237.722,5.364,-40.865,-179.316,5.252,148.701
C04694=1237.727,5.115,-40.850,-179.319,5.252,148.702
C04695=1237.733,4.865,-40.835,-179.322,5.251,148.703
C04696=1237.737,4.616,-40.820,-179.324,5.251,148.704
C04697=1237.742,4.366,-40.806,-179.326,5.251,148.704
C04698=1237.748,4.097,-40.789,-179.329,5.250,148.705
C04699=1237.753,3.828,-40.774,-179.332,5.250,148.706
C04700=1237.758,3.560,-40.758,-179.335,5.250,148.706
C04701=1237.764,3.291,-40.742,-179.337,5.250,148.707
C04702=1237.769,3.041,-40.727,-179.340,5.249,148.708
C04703=1237.774,2.792,-40.712,-179.342,5.249,148.709
C04704=1237.778,2.543,-40.697,-179.344,5.249,148.709
C04705=1237.784,2.293,-40.683,-179.347,5.249,148.710
C04706=1237.789,2.043,-40.668,-179.350,5.248,148.711
C04707=1237.794,1.794,-40.653,-179.352,5.248,148.711
C04708=1237.799,1.544,-40.639,-179.355,5.248,148.712
C04709=1237.803,1.295,-40.624,-179.357,5.248,148.713
C04710=1237.809,1.045,-40.609,-179.360,5.247,148.714
C04711=1237.814,0.795,-40.595,-179.362,5.247,148.714
C04712=1237.819,0.546,-40.580,-179.365,5.247,148.715
C04713=1237.824,0.297,-40.566,-179.368,5.246,148.716
C04714=1237.829,0.047,-40.551,-179.370,5.247,148.716
C04715=1237.834,-0.203,-40.536,-179.372,5.246,148.717
C04716=1237.839,-0.452,-40.521,-179.375,5.246,148.718
C04717=1237.844,-0.702,-40.507,-179.377,5.246,148.718
C04718=1237.848,-0.951,-40.492,-179.380,5.245,148.719
C04719=1237.853,-1.201,-40.478,-179.382,5.245,148.720
C04720=1237.859,-1.451,-40.463,-179.384,5.245,148.721
C04721=1237.864,-1.699,-40.448,-179.387,5.244,148.721
C04722=1237.869,-1.949,-40.434,-179.390,5.244,148.722
C04723=1237.874,-2.199,-40.420,-179.392,5.244,148.723
C04724=1237.879,-2.448,-40.406,-179.394,5.244,148.723
C04725=1237.884,-2.697,-40.391,-179.397,5.243,148.724
C04726=1237.889,-2.947,-40.376,-179.400,5.244,148.725
C04727=1237.894,-3.197,-40.362,-179.402,5.243,148.726
C04728=1237.899,-3.447,-40.347,-179.405,5.243,148.726
C04729=1237.904,-3.696,-40.332,-179.407,5.243,148.727
C04730=1237.909,-3.946,-40.318,-179.410,5.243,148.728
C04731=1237.914,-4.195,-40.304,-179.412,5.242,148.728
C04732=1237.920,-4.444,-40.290,-179.414,5.242,148.729
C04733=1237.924,-4.694,-40.275,-179.417,5.242,148.730
C04734=1237.929,-4.943,-40.260,-179.420,5.241,148.730
C04735=1237.934,-5.193,-40.246,-179.422,5.241,148.731
C04736=1237.939,-5.443,-40.232,-179.424,5.241,148.732
C04737=1237.944,-5.692,-40.218,-179.427,5.240,148.732
C04738=1237.949,-5.942,-40.203,-179.429,5.241,148.733
C04739=1237.954,-6.191,-40.188,-179.432,5.240,148.734
C04740=1237.960,-6.440,-40.174,-179.435,5.240,148.735
C04741=1237.965,-6.690,-40.159,-179.437,5.240,148.735
C04742=1237.970,-6.940,-40.145,-179.439,5.239,148.736
C04743=1237.975,-7.190,-40.131,-179.442,5.239,148.737
C04744=1237.980,-7.439,-40.117,-179.444,5.240,148.738
C04745=1237.985,-7.689,-40.102,-179.447,5.239,148.738
C04746=1237.989,-7.938,-40.087,-179.450,5.238,148.739
C04747=1237.995,-8.187,-40.073,-179.452,5.239,148.740
C04748=1238.000,-8.437,-40.059,-179.455,5.238,148.740
C04749=1238.005,-8.687,-40.045,-179.457,5.238,148.741
C04750=1238.010,-8.936,-40.031,-179.459,5.238,148.742
C04751=1238.015,-9.186,-40.016,-179.462,5.237,148.742
C04752=1238.020,-9.436,-40.002,-179.465,5.237,148.743
C04753=1238.025,-9.685,-39.988,-179.467,5.237,148.744
C04754=1238.030,-9.934,-39.974,-179.469,5.237,148.744
C04755=1238.035,-10.184,-39.960,-179.472,5.236,148.745
C04756=1238.040,-10.434,-39.945,-179.474,5.236,148.746
C04757=1238.045,-10.684,-39.931,-179.477,5.236,148.747
C04758=1238.050,-10.932,-39.918,-179.479,5.237,148.747
C04759=1238.055,-11.182,-39.903,-179.482,5.236,148.748
C04760=1238.060,-11.432,-39.889,-179.485,5.235,148.749
C04761=1238.065,-11.681,-39.875,-179.487,5.236,148.750
C04762=1238.070,-11.931,-39.861,-179.489,5.235,148.750
C04763=1238.075,-12.180,-39.847,-179.492,5.235,148.751
C04764=1238.080,-12.430,-39.832,-179.494,5.235,148.752
C04765=1238.085,-12.680,-39.818,-179.497,5.234,148.752
C04766=1238.090,-12.929,-39.804,-179.499,5.234,148.753
C04767=1238.096,-13.178,-39.790,-179.501,5.234,148.754
C04768=1238.101,-13.428,-39.776,-179.504,5.234,148.754
C04769=1238.106,-13.678,-39.761,-179.507,5.233,148.755
C04770=1238.110,-13.927,-39.748,-179.509,5.233,148.756
C04771=1238.115,-14.176,-39.734,-179.512,5.233,148.757
C04772=1238.120,-14.426,-39.720,-179.514,5.234,148.757
C04773=1238.125,-14.675,-39.705,-179.517,5.233,148.758
C04774=1238.131,-14.926,-39.692,-179.519,5.233,148.759
C04775=1238.136,-15.175,-39.678,-179.521,5.233,148.760
C04776=1238.141,-15.425,-39.664,-179.524,5.232,148.760
C04777=1238.146,-15.674,-39.649,-179.527,5.232,148.761
C04778=1238.150,-15.924,-39.636,-179.529,5.232,148.762
C04779=1238.156,-16.173,-39.622,-179.532,5.232,148.762
C04780=1238.161,-16.422,-39.607,-179.534,5.231,148.763
C04781=1238.166,-16.672,-39.593,-179.536,5.231,148.764
C04782=1238.171,-16.922,-39.580,-179.539,5.231,148.764
C04783=1238.177,-17.171,-39.566,-179.541,5.231,148.765
C04784=1238.181,-17.421,-39.552,-179.544,5.231,148.766
C04785=1238.186,-17.671,-39.538,-179.547,5.230,148.767
C04786=1238.191,-17.920,-39.524,-179.549,5.231,148.767
C04787=1238.196,-18.170,-39.510,-179.552,5.230,148.768
C04788=1238.201,-18.420,-39.496,-179.554,5.230,148.769
C04789=1238.206,-18.668,-39.483,-179.556,5.230,148.769
C04790=1238.211,-18.918,-39.468,-179.559,5.229,148.770
C04791=1238.216,-19.168,-39.454,-179.561,5.230,148.771
C04792=1238.222,-19.417,-39.441,-179.564,5.229,148.772
C04793=1238.227,-19.667,-39.427,-179.566,5.229,148.772
C04794=1238.231,-19.916,-39.413,-179.568,5.229,148.773
C04795=1238.237,-20.165,-39.399,-179.571,5.229,148.774
C04796=1238.242,-20.416,-39.385,-179.574,5.228,148.774
C04797=1238.247,-20.665,-39.371,-179.576,5.228,148.775
C04798=1238.252,-20.914,-39.358,-179.579,5.228,148.776
C04799=1238.257,-21.165,-39.344,-179.581,5.228,148.777
C04800=1238.262,-21.414,-39.330,-179.584,5.228,148.777
C04801=1238.268,-21.663,-39.316,-179.586,5.227,148.778
C04802=1238.272,-21.932,-39.302,-179.588,5.228,148.779
C04803=1238.278,-22.202,-39.287,-179.591,5.227,148.779
C04804=1238.283,-22.471,-39.272,-179.594,5.227,148.780
C04805=1238.289,-22.741,-39.257,-179.597,5.226,148.781
C04806=1238.294,-22.990,-39.244,-179.599,5.227,148.782
C04807=1238.299,-23.240,-39.230,-179.602,5.226,148.782
C04808=1238.304,-23.489,-39.216,-179.604,5.227,148.783
C04809=1238.309,-23.739,-39.202,-179.606,5.226,148.784
C04810=1238.314,-23.988,-39.189,-179.610,5.226,148.785
C04811=1238.319,-24.237,-39.175,-179.612,5.226,148.785
C04812=1238.324,-24.488,-39.161,-179.614,5.226,148.786
C04813=1238.329,-24.737,-39.148,-179.616,5.226,148.787
C04814=1238.335,-24.987,-39.134,-179.619,5.225,148.788
C04815=1238.340,-25.236,-39.120,-179.622,5.225,148.788
C04816=1238.344,-25.485,-39.107,-179.624,5.225,148.789
C04817=1238.350,-25.735,-39.093,-179.626,5.225,148.790
C04818=1238.354,-25.985,-39.080,-179.629,5.225,148.790
C04819=1238.360,-26.234,-39.066,-179.631,5.225,148.791
C04820=1238.365,-26.484,-39.052,-179.634,5.224,148.792
C04821=1238.370,-26.734,-39.039,-179.636,5.224,148.792
C04822=1238.375,-26.983,-39.025,-179.639,5.224,148.793
C04823=1238.381,-27.233,-39.012,-179.641,5.224,148.794
C04824=1238.385,-27.482,-38.998,-179.644,5.224,148.795
C04825=1238.390,-27.733,-38.985,-179.647,5.223,148.795
C04826=1238.395,-27.981,-38.971,-179.649,5.224,148.796
C04827=1238.400,-28.232,-38.958,-179.651,5.223,148.797
C04828=1238.406,-28.481,-38.944,-179.653,5.224,148.798
C04829=1238.410,-28.731,-38.931,-179.656,5.223,148.798
C04830=1238.416,-28.980,-38.917,-179.659,5.223,148.799
C04831=1238.420,-29.230,-38.904,-179.661,5.223,148.800
C04832=1238.426,-29.479,-38.890,-179.663,5.222,148.800
C04833=1238.430,-29.729,-38.877,-179.666,5.223,148.801
C04834=1238.436,-29.978,-38.863,-179.668,5.222,148.802
C04835=1238.440,-30.228,-38.850,-179.671,5.222,148.803
C04836=1238.445,-30.477,-38.836,-179.673,5.222,148.803
C04837=1238.451,-30.727,-38.823,-179.676,5.222,148.804
C04838=1238.456,-30.977,-38.810,-179.678,5.222,148.805
C04839=1238.461,-31.226,-38.796,-179.681,5.222,148.805
C04840=1238.466,-31.476,-38.783,-179.683,5.221,148.806
C04841=1238.471,-31.725,-38.769,-179.686,5.221,148.807
C04842=1238.476,-31.975,-38.756,-179.688,5.221,148.808
C04843=1238.482,-32.225,-38.743,-179.690,5.221,148.808
C04844=1238.486,-32.474,-38.729,-179.693,5.221,148.809
C04845=1238.492,-32.724,-38.716,-179.695,5.221,148.810
C04846=1238.496,-32.973,-38.702,-179.698,5.221,148.811
C04847=1238.502,-33.223,-38.689,-179.701,5.220,148.811
C04848=1238.506,-33.473,-38.676,-179.703,5.221,148.812
C04849=1238.512,-33.722,-38.662,-179.706,5.220,148.813
C04850=1238.517,-33.972,-38.649,-179.708,5.220,148.813
C04851=1238.522,-34.221,-38.637,-179.710,5.220,148.814
C04852=1238.527,-34.471,-38.622,-179.713,5.219,148.815
C04853=1238.532,-34.720,-38.610,-179.715,5.220,148.815
C04854=1238.538,-34.970,-38.597,-179.718,5.219,148.816
C04855=1238.542,-35.220,-38.584,-179.720,5.219,148.817
C04856=1238.548,-35.469,-38.570,-179.723,5.219,148.818
C04857=1238.552,-35.719,-38.557,-179.725,5.219,148.818
C04858=1238.558,-35.969,-38.544,-179.728,5.219,148.819
C04859=1238.562,-36.218,-38.530,-179.730,5.219,148.820
C04860=1238.567,-36.467,-38.517,-179.733,5.219,148.821
C04861=1238.573,-36.718,-38.504,-179.735,5.218,148.821
C04862=1238.578,-36.967,-38.491,-179.737,5.219,148.822
C04863=1238.583,-37.216,-38.477,-179.740,5.218,148.823
C04864=1238.588,-37.466,-38.464,-179.742,5.219,148.823
C04865=1238.593,-37.715,-38.452,-179.745,5.218,148.824
C04866=1238.598,-37.966,-38.438,-179.747,5.218,148.825
C04867=1238.603,-38.215,-38.426,-179.749,5.218,148.825
C04868=1238.608,-38.465,-38.411,-179.752,5.217,148.826
C04869=1238.613,-38.714,-38.399,-179.755,5.218,148.827
C04870=1238.619,-38.963,-38.386,-179.757,5.218,148.828
C04871=1238.624,-39.214,-38.372,-179.759,5.218,148.829
C04872=1238.629,-39.463,-38.360,-179.762,5.217,148.829
C04873=1238.634,-39.713,-38.347,-179.765,5.217,148.830
C04874=1238.639,-39.962,-38.333,-179.767,5.217,148.831
C04875=1238.644,-40.211,-38.320,-179.770,5.217,148.831
C04876=1238.649,-40.461,-38.307,-179.772,5.217,148.832
C04877=1238.655,-40.711,-38.294,-179.774,5.216,148.833
C04878=1238.659,-40.961,-38.281,-179.776,5.217,148.833
C04879=1238.664,-41.210,-38.269,-179.779,5.216,148.834
C04880=1238.670,-41.460,-38.255,-179.782,5.216,148.835
C04881=1238.675,-41.710,-38.243,-179.784,5.216,148.836
C04882=1238.679,-41.959,-38.229,-179.787,5.216,148.836
C04883=1238.685,-42.208,-38.216,-179.789,5.216,148.837
C04884=1238.690,-42.458,-38.203,-179.792,5.216,148.838
C04885=1238.695,-42.707,-38.190,-179.794,5.216,148.839
C04886=1238.700,-42.957,-38.178,-179.796,5.216,148.839
C04887=1238.705,-43.207,-38.164,-179.799,5.215,148.840
C04888=1238.710,-43.456,-38.152,-179.801,5.215,148.841
C04889=1238.715,-43.706,-38.139,-179.804,5.215,148.841
C04890=1238.720,-43.956,-38.126,-179.806,5.215,148.842
C04891=1238.726,-44.205,-38.113,-179.809,5.215,148.843
C04892=1238.730,-44.455,-38.100,-179.811,5.215,148.843
C04893=1238.736,-44.705,-38.087,-179.814,5.215,148.844
C04894=1238.741,-44.954,-38.075,-179.816,5.215,148.845
C04895=1238.746,-45.204,-38.061,-179.819,5.215,148.846
C04896=1238.751,-45.454,-38.049,-179.821,5.214,148.847
C04897=1238.756,-45.703,-38.036,-179.823,5.214,148.847
C04898=1238.761,-45.952,-38.023,-179.826,5.214,148.848
C04899=1238.767,-46.203,-38.010,-179.828,5.214,148.849
C04900=1238.772,-46.452,-37.997,-179.831,5.214,148.849
C04901=1238.777,-46.701,-37.985,-179.833,5.214,148.850
C04902=1238.781,-46.951,-37.972,-179.835,5.214,148.851
C04903=1238.787,-47.201,-37.959,-179.838,5.214,148.851
C04904=1238.792,-47.450,-37.946,-179.841,5.214,148.852
C04905=1238.797,-47.700,-37.933,-179.843,5.214,148.853
C04906=1238.802,-47.969,-37.920,-179.845,5.214,148.854
C04907=1238.808,-48.239,-37.905,-179.848,5.213,148.854
C04908=1238.813,-48.509,-37.892,-179.851,5.213,148.855
C04909=1238.819,-48.778,-37.878,-179.853,5.213,148.856
C04910=1238.824,-49.029,-37.865,-179.856,5.213,148.857
C04911=1238.830,-49.278,-37.853,-179.858,5.213,148.858
C04912=1238.835,-49.528,-37.840,-179.861,5.213,148.858
C04913=1238.840,-49.777,-37.828,-179.863,5.213,148.859
C04914=1238.844,-50.027,-37.815,-179.866,5.212,148.860
C04915=1238.849,-50.276,-37.802,-179.868,5.213,148.860
C04916=1238.855,-50.526,-37.789,-179.871,5.213,148.861
C04917=1238.860,-50.775,-37.777,-179.874,5.212,148.862
C04918=1238.865,-51.026,-37.764,-179.876,5.212,148.863
C04919=1238.870,-51.275,-37.751,-179.878,5.212,148.863
C04920=1238.875,-51.525,-37.739,-179.880,5.212,148.864
C04921=1238.881,-51.774,-37.726,-179.883,5.212,148.865
C04922=1238.885,-52.024,-37.713,-179.885,5.212,148.865
C04923=1238.891,-52.274,-37.701,-179.888,5.212,148.866
C04924=1238.896,-52.523,-37.689,-179.890,5.212,148.867
C04925=1238.901,-52.772,-37.676,-179.893,5.211,148.868
C04926=1238.905,-53.023,-37.663,-179.895,5.212,148.868
C04927=1238.910,-53.272,-37.651,-179.897,5.211,148.869
C04928=1238.916,-53.522,-37.639,-179.900,5.212,148.870
C04929=1238.921,-53.771,-37.626,-179.903,5.212,148.871
C04930=1238.926,-54.020,-37.614,-179.905,5.211,148.871
C04931=1238.931,-54.270,-37.601,-179.907,5.211,148.872
C04932=1238.936,-54.520,-37.589,-179.910,5.211,148.873
C04933=1238.942,-54.770,-37.575,-179.912,5.211,148.873
C04934=1238.947,-55.019,-37.563,-179.915,5.211,148.874
C04935=1238.952,-55.269,-37.551,-179.917,5.211,148.875
C04936=1238.957,-55.519,-37.538,-179.919,5.211,148.876
C04937=1238.962,-55.769,-37.525,-179.922,5.211,148.876
C04938=1238.967,-56.018,-37.513,-179.924,5.210,148.877
C04939=1238.973,-56.268,-37.501,-179.926,5.211,148.878
C04940=1238.978,-56.517,-37.488,-179.929,5.211,148.879
C04941=1238.983,-56.766,-37.476,-179.932,5.211,148.879
C04942=1238.988,-57.017,-37.463,-179.934,5.210,148.880
C04943=1238.993,-57.266,-37.451,-179.936,5.211,148.881
C04944=1238.997,-57.515,-37.439,-179.939,5.210,148.881
C04945=1239.003,-57.765,-37.427,-179.941,5.211,148.882
C04946=1239.008,-58.015,-37.414,-179.944,5.210,148.883
C04947=1239.013,-58.265,-37.403,-179.946,5.210,148.884
C04948=1239.018,-58.515,-37.390,-179.948,5.210,148.884
C04949=1239.023,-58.764,-37.377,-179.951,5.209,148.885
C04950=1239.028,-59.014,-37.365,-179.953,5.210,148.886
C04951=1239.033,-59.263,-37.352,-179.956,5.209,148.886
C04952=1239.039,-59.513,-37.340,-179.958,5.210,148.887
C04953=1239.044,-59.762,-37.328,-179.961,5.209,148.888
C04954=1239.049,-60.012,-37.315,-179.963,5.210,148.889
C04955=1239.054,-60.262,-37.303,-179.966,5.209,148.889
C04956=1239.059,-60.512,-37.291,-179.968,5.210,148.890
C04957=1239.065,-60.762,-37.279,-179.971,5.209,148.891
C04958=1239.070,-61.011,-37.266,-179.973,5.209,148.892
C04959=1239.075,-61.261,-37.254,-179.975,5.209,148.892
C04960=1239.079,-61.510,-37.242,-179.978,5.209,148.893
C04961=1239.085,-61.759,-37.230,-179.980,5.209,148.894
C04962=1239.090,-62.009,-37.218,-179.982,5.209,148.894
C04963=1239.095,-62.259,-37.205,-179.985,5.209,148.895
C04964=1239.100,-62.509,-37.193,-179.987,5.209,148.896
C04965=1239.105,-62.758,-37.180,-179.990,5.208,148.896
C04966=1239.111,-63.008,-37.168,-179.992,5.209,148.897
C04967=1239.116,-63.258,-37.156,-179.995,5.209,148.898
C04968=1239.120,-63.507,-37.144,-179.997,5.209,148.899
C04969=1239.125,-63.757,-37.132,-180.000,5.209,148.900
C04970=1239.131,-64.007,-37.120,179.998,5.208,148.900
C04971=1239.136,-64.257,-37.108,179.996,5.208,148.901
C04972=1239.141,-64.506,-37.095,179.993,5.208,148.902
C04973=1239.147,-64.756,-37.084,179.991,5.208,148.902
C04974=1239.151,-65.005,-37.072,179.988,5.208,148.903
C04975=1239.157,-65.255,-37.060,179.986,5.208,148.904
C04976=1239.162,-65.504,-37.047,179.983,5.208,148.904
C04977=1239.167,-65.754,-37.035,179.981,5.208,148.905
C04978=1239.173,-66.004,-37.023,179.979,5.207,148.906
C04979=1239.178,-66.253,-37.011,179.976,5.208,148.907
C04980=1239.182,-66.504,-36.999,179.973,5.208,148.908
C04981=1239.187,-66.753,-36.986,179.971,5.208,148.908
C04982=1239.192,-67.003,-36.975,179.969,5.208,148.909
C04983=1239.198,-67.253,-36.963,179.966,5.208,148.910
C04984=1239.202,-67.502,-36.951,179.964,5.207,148.910
C04985=1239.208,-67.752,-36.939,179.962,5.208,148.911
C04986=1239.213,-68.002,-36.927,179.959,5.207,148.912
C04987=1239.218,-68.251,-36.914,179.957,5.208,148.912
C04988=1239.224,-68.501,-36.902,179.954,5.207,148.913
C04989=1239.228,-68.751,-36.891,179.952,5.207,148.914
C04990=1239.233,-69.000,-36.879,179.950,5.207,148.915
C04991=1239.239,-69.250,-36.867,179.947,5.207,148.915
C04992=1239.244,-69.499,-36.855,179.945,5.207,148.916
C04993=1239.249,-69.749,-36.843,179.943,5.207,148.917
C04994=1239.254,-69.999,-36.831,179.939,5.207,148.918
C04995=1239.260,-70.249,-36.819,179.937,5.207,148.918
C04996=1239.264,-70.498,-36.807,179.935,5.207,148.919
C04997=1239.269,-70.748,-36.795,179.933,5.207,148.920
C04998=1239.275,-70.997,-36.783,179.930,5.207,148.921
C04999=1239.280,-71.247,-36.771,179.928,5.207,148.921
C05000=1239.285,-71.496,-36.760,179.925,5.207,148.922
C05001=1239.291,-71.746,-36.748,179.923,5.207,148.923
C05002=1239.296,-71.996,-36.736,179.920,5.206,148.923
C05003=1239.301,-72.245,-36.725,179.918,5.207,148.924
C05004=1239.306,-72.495,-36.712,179.916,5.206,148.925
C05005=1239.311,-72.744,-36.700,179.914,5.207,148.925
C05006=1239.316,-72.994,-36.689,179.911,5.206,148.926
C05007=1239.321,-73.244,-36.677,179.909,5.206,148.927
C05008=1239.327,-73.494,-36.665,179.906,5.206,148.928
C05009=1239.331,-73.743,-36.653,179.904,5.207,148.929
C05010=1239.337,-74.014,-36.641,179.901,5.206,148.929
C05011=1239.343,-74.284,-36.628,179.899,5.207,148.930
C05012=1239.348,-74.554,-36.615,179.896,5.206,148.931
C05013=1239.353,-74.824,-36.602,179.893,5.206,148.932
C05014=1239.359,-75.074,-36.591,179.891,5.206,148.932
C05015=1239.365,-75.323,-36.579,179.888,5.206,148.933
C05016=1239.370,-75.573,-36.568,179.886,5.206,148.934
C05017=1239.375,-75.822,-36.555,179.883,5.206,148.934
C05018=1239.380,-76.072,-36.543,179.881,5.206,148.935
C05019=1239.385,-76.322,-36.532,179.879,5.206,148.936
C05020=1239.390,-76.572,-36.520,179.877,5.206,148.937
C05021=1239.395,-76.822,-36.509,179.874,5.205,148.937
C05022=1239.400,-77.071,-36.497,179.872,5.206,148.938
C05023=1239.405,-77.321,-36.485,179.869,5.205,148.939
C05024=1239.411,-77.570,-36.474,179.867,5.206,148.939
C05025=1239.417,-77.820,-36.462,179.864,5.205,148.940
C05026=1239.421,-78.070,-36.451,179.862,5.206,148.941
C05027=1239.427,-78.320,-36.439,179.859,5.205,148.942
C05028=1239.431,-78.569,-36.428,179.857,5.206,148.942
C05029=1239.436,-78.819,-36.415,179.854,5.205,148.943
C05030=1239.441,-79.068,-36.404,179.852,5.206,148.944
C05031=1239.447,-79.318,-36.392,179.850,5.205,148.945
C05032=1239.452,-79.567,-36.381,179.848,5.206,148.945
C05033=1239.457,-79.817,-36.369,179.845,5.205,148.946
C05034=1239.463,-80.067,-36.357,179.843,5.205,148.947
C05035=1239.467,-80.317,-36.346,179.840,5.205,148.947
C05036=1239.473,-80.567,-36.334,179.838,5.205,148.948
C05037=1239.478,-80.816,-36.323,179.835,5.205,148.949
C05038=1239.483,-81.066,-36.311,179.833,5.205,148.950
C05039=1239.488,-81.315,-36.300,179.831,5.205,148.950
C05040=1239.494,-81.565,-36.288,179.828,5.205,148.951
C05041=1239.498,-81.815,-36.277,179.826,5.205,148.952
C05042=1239.504,-82.065,-36.265,179.824,5.205,148.952
C05043=1239.509,-82.315,-36.254,179.822,5.205,148.953
C05044=1239.514,-82.565,-36.243,179.819,5.205,148.954
C05045=1239.520,-82.814,-36.231,179.816,5.205,148.955
C05046=1239.524,-83.063,-36.220,179.814,5.205,148.955
C05047=1239.530,-83.313,-36.208,179.812,5.205,148.956
C05048=1239.534,-83.563,-36.197,179.809,5.205,148.957
C05049=1239.540,-83.813,-36.185,179.807,5.205,148.958
C05050=1239.545,-84.062,-36.174,179.804,5.205,148.958
C05051=1239.551,-84.312,-36.162,179.802,5.205,148.959
C05052=1239.555,-84.561,-36.151,179.799,5.205,148.960
C05053=1239.560,-84.811,-36.140,179.797,5.205,148.960
C05054=1239.565,-85.061,-36.128,179.795,5.205,148.961
C05055=1239.571,-85.311,-36.118,179.793,5.205,148.962
C05056=1239.576,-85.560,-36.106,179.790,5.204,148.963
C05057=1239.581,-85.810,-36.094,179.788,5.205,148.963
C05058=1239.586,-86.060,-36.083,179.785,5.204,148.964
C05059=1239.591,-86.310,-36.071,179.783,5.205,148.965
C05060=1239.596,-86.559,-36.060,179.780,5.204,148.965
C05061=1239.602,-86.809,-36.049,179.778,5.204,148.966
C05062=1239.607,-87.059,-36.038,179.776,5.204,148.967
C05063=1239.612,-87.308,-36.027,179.773,5.204,148.968
C05064=1239.618,-87.558,-36.015,179.771,5.205,148.968
C05065=1239.622,-87.807,-36.004,179.769,5.204,148.969
C05066=1239.628,-88.058,-35.993,179.767,5.205,148.970
C05067=1239.633,-88.307,-35.981,179.764,5.204,148.970
C05068=1239.638,-88.556,-35.970,179.762,5.204,148.971
C05069=1239.643,-88.806,-35.958,179.759,5.204,148.972
C05070=1239.648,-89.056,-35.947,179.757,5.205,148.973
C05071=1239.653,-89.306,-35.937,179.754,5.204,148.973
C05072=1239.659,-89.555,-35.925,179.752,5.205,148.974
C05073=1239.664,-89.805,-35.914,179.749,5.204,148.975
C05074=1239.669,-90.055,-35.903,179.747,5.205,148.976
C05075=1239.674,-90.305,-35.891,179.744,5.204,148.976
C05076=1239.680,-90.554,-35.880,179.742,5.204,148.977
C05077=1239.684,-90.804,-35.869,179.740,5.204,148.978
C05078=1239.689,-91.054,-35.859,179.738,5.204,148.978
C05079=1239.695,-91.303,-35.847,179.735,5.204,148.979
C05080=1239.700,-91.553,-35.836,179.733,5.204,148.980
C05081=1239.705,-91.802,-35.824,179.730,5.204,148.981
C05082=1239.711,-92.052,-35.814,179.728,5.204,148.981
C05083=1239.716,-92.302,-35.802,179.726,5.204,148.982
C05084=1239.720,-92.552,-35.791,179.723,5.204,148.983
C05085=1239.725,-92.802,-35.780,179.721,5.204,148.983
C05086=1239.731,-93.051,-35.769,179.718,5.204,148.984
C05087=1239.736,-93.301,-35.758,179.716,5.204,148.985
C05088=1239.741,-93.551,-35.747,179.714,5.204,148.986
C05089=1239.747,-93.800,-35.736,179.712,5.204,148.986
C05090=1239.752,-94.050,-35.725,179.709,5.204,148.987
C05091=1239.757,-94.300,-35.714,179.707,5.204,148.988
C05092=1239.762,-94.549,-35.703,179.704,5.204,148.988
C05093=1239.767,-94.799,-35.692,179.702,5.204,148.989
C05094=1239.773,-95.049,-35.680,179.699,5.203,148.990
C05095=1239.778,-95.299,-35.670,179.697,5.204,148.991
C05096=1239.783,-95.548,-35.659,179.695,5.203,148.991
C05097=1239.788,-95.797,-35.648,179.693,5.204,148.992
C05098=1239.794,-96.048,-35.637,179.690,5.204,148.993
C05099=1239.799,-96.297,-35.625,179.688,5.204,148.993
C05100=1239.804,-96.547,-35.615,179.686,5.204,148.994
C05101=1239.809,-96.797,-35.604,179.683,5.203,148.995
C05102=1239.814,-97.047,-35.593,179.681,5.204,148.996
C05103=1239.820,-97.296,-35.582,179.678,5.203,148.996
C05104=1239.825,-97.546,-35.571,179.676,5.204,148.997
C05105=1239.830,-97.796,-35.560,179.673,5.203,148.998
C05106=1239.835,-98.045,-35.549,179.671,5.204,148.998
C05107=1239.840,-98.295,-35.538,179.669,5.203,148.999
C05108=1239.845,-98.544,-35.528,179.667,5.203,149.000
C05109=1239.851,-98.795,-35.516,179.664,5.203,149.001
C05110=1239.856,-99.044,-35.505,179.662,5.203,149.001
C05111=1239.861,-99.294,-35.495,179.660,5.204,149.002
C05112=1239.866,-99.544,-35.484,179.657,5.204,149.003
C05113=1239.871,-99.793,-35.473,179.654,5.204,149.004
C05114=1239.877,-100.064,-35.461,179.652,5.204,149.004
C05115=1239.882,-100.335,-35.450,179.649,5.203,149.005
C05116=1239.888,-100.605,-35.438,179.647,5.203,149.006
C05117=1239.894,-100.876,-35.426,179.644,5.203,149.007
C05118=1239.899,-101.127,-35.416,179.642,5.204,149.007
C05119=1239.904,-101.376,-35.405,179.639,5.203,149.008
C05120=1239.909,-101.626,-35.394,179.637,5.204,149.009
C05121=1239.915,-101.875,-35.383,179.634,5.203,149.010
C05122=1239.920,-102.125,-35.373,179.632,5.204,149.010
C05123=1239.925,-102.375,-35.362,179.630,5.204,149.011
C05124=1239.930,-102.624,-35.351,179.627,5.203,149.012
C05125=1239.935,-102.874,-35.340,179.625,5.204,149.012
C05126=1239.940,-103.123,-35.330,179.623,5.203,149.013
C05127=1239.945,-103.374,-35.319,179.621,5.204,149.014
C05128=1239.951,-103.623,-35.309,179.618,5.203,149.015
C05129=1239.956,-103.873,-35.297,179.616,5.204,149.015
C05130=1239.962,-104.123,-35.287,179.613,5.203,149.016
C05131=1239.967,-104.373,-35.276,179.611,5.204,149.017
C05132=1239.972,-104.622,-35.265,179.608,5.203,149.017
C05133=1239.977,-104.872,-35.255,179.606,5.203,149.018
C05134=1239.982,-105.122,-35.244,179.604,5.204,149.019
C05135=1239.987,-105.371,-35.233,179.601,5.203,149.020
C05136=1239.992,-105.621,-35.222,179.599,5.204,149.020
C05137=1239.998,-105.871,-35.212,179.597,5.203,149.021
C05138=1240.003,-106.121,-35.201,179.595,5.204,149.022
C05139=1240.008,-106.370,-35.191,179.592,5.203,149.022
C05140=1240.013,-106.620,-35.180,179.590,5.204,149.023
C05141=1240.019,-106.870,-35.170,179.587,5.203,149.024
C05142=1240.024,-107.120,-35.159,179.585,5.203,149.025
C05143=1240.029,-107.369,-35.148,179.582,5.203,149.025
C05144=1240.034,-107.619,-35.138,179.580,5.203,149.026
C05145=1240.040,-107.868,-35.127,179.579,5.203,149.026
C05146=1240.045,-108.119,-35.116,179.576,5.203,149.027
C05147=1240.050,-108.368,-35.106,179.574,5.203,149.028
C05148=1240.055,-108.618,-35.096,179.571,5.203,149.029
C05149=1240.061,-108.868,-35.085,179.569,5.203,149.029
C05150=1240.065,-109.116,-35.075,179.566,5.203,149.030
C05151=1240.070,-109.367,-35.065,179.564,5.203,149.031
C05152=1240.076,-109.616,-35.054,179.562,5.203,149.031
C05153=1240.081,-109.867,-35.044,179.560,5.203,149.032
C05154=1240.086,-110.116,-35.034,179.557,5.203,149.033
C05155=1240.091,-110.366,-35.022,179.555,5.203,149.034
C05156=1240.097,-110.615,-35.012,179.553,5.203,149.034
C05157=1240.102,-110.865,-35.001,179.550,5.203,149.035
C05158=1240.107,-111.115,-34.991,179.548,5.203,149.036
C05159=1240.112,-111.365,-34.981,179.545,5.203,149.036
C05160=1240.118,-111.615,-34.970,179.543,5.203,149.037
C05161=1240.123,-111.864,-34.960,179.540,5.203,149.038
C05162=1240.128,-112.114,-34.950,179.538,5.203,149.039
C05163=1240.133,-112.363,-34.939,179.536,5.203,149.039
C05164=1240.138,-112.613,-34.929,179.534,5.203,149.040
C05165=1240.144,-112.863,-34.919,179.532,5.203,149.041
C05166=1240.149,-113.113,-34.908,179.529,5.203,149.041
C05167=1240.154,-113.363,-34.898,179.527,5.203,149.042
C05168=1240.160,-113.612,-34.888,179.524,5.203,149.043
C05169=1240.165,-113.863,-34.877,179.522,5.203,149.044
C05170=1240.169,-114.111,-34.867,179.519,5.203,149.044
C05171=1240.174,-114.361,-34.856,179.517,5.203,149.045
C05172=1240.180,-114.611,-34.846,179.514,5.203,149.046
C05173=1240.186,-114.861,-34.836,179.512,5.203,149.047
C05174=1240.191,-115.111,-34.825,179.510,5.203,149.047
C05175=1240.196,-115.360,-34.815,179.508,5.203,149.048
C05176=1240.201,-115.611,-34.804,179.506,5.203,149.049
C05177=1240.206,-115.860,-34.795,179.503,5.203,149.049
C05178=1240.212,-116.109,-34.785,179.501,5.203,149.050
C05179=1240.217,-116.360,-34.774,179.498,5.203,149.051
C05180=1240.222,-116.609,-34.764,179.496,5.203,149.052
C05181=1240.228,-116.859,-34.754,179.493,5.203,149.052
C05182=1240.232,-117.109,-34.744,179.492,5.203,149.053
C05183=1240.238,-117.358,-34.733,179.490,5.203,149.053
C05184=1240.243,-117.608,-34.723,179.487,5.203,149.054
C05185=1240.248,-117.858,-34.713,179.485,5.203,149.055
C05186=1240.253,-118.107,-34.703,179.482,5.203,149.056
C05187=1240.258,-118.357,-34.692,179.480,5.203,149.056
C05188=1240.264,-118.607,-34.682,179.477,5.202,149.057
C05189=1240.269,-118.856,-34.672,179.475,5.203,149.058
C05190=1240.274,-119.106,-34.662,179.473,5.202,149.058
C05191=1240.279,-119.356,-34.652,179.471,5.203,149.059
C05192=1240.285,-119.606,-34.642,179.468,5.203,149.060
C05193=1240.290,-119.856,-34.631,179.466,5.203,149.061
C05194=1240.295,-120.105,-34.621,179.464,5.203,149.061
C05195=1240.301,-120.355,-34.612,179.461,5.203,149.062
C05196=1240.306,-120.605,-34.601,179.459,5.203,149.063
C05197=1240.311,-120.855,-34.591,179.456,5.203,149.063
C05198=1240.316,-121.104,-34.581,179.454,5.203,149.064
C05199=1240.321,-121.354,-34.571,179.452,5.203,149.065
C05200=1240.327,-121.604,-34.561,179.449,5.203,149.066
C05201=1240.332,-121.853,-34.551,179.447,5.203,149.066
C05202=1240.337,-122.103,-34.540,179.445,5.202,149.067
C05203=1240.342,-122.353,-34.530,179.443,5.203,149.068
C05204=1240.348,-122.603,-34.521,179.440,5.202,149.068
C05205=1240.353,-122.852,-34.511,179.438,5.203,149.069
C05206=1240.358,-123.103,-34.501,179.435,5.202,149.070
C05207=1240.363,-123.352,-34.490,179.433,5.203,149.070
C05208=1240.368,-123.601,-34.481,179.431,5.203,149.071
C05209=1240.373,-123.852,-34.470,179.429,5.203,149.072
C05210=1240.379,-124.102,-34.461,179.426,5.203,149.073
C05211=1240.384,-124.351,-34.451,179.424,5.203,149.073
C05212=1240.390,-124.601,-34.441,179.422,5.203,149.074
C05213=1240.394,-124.851,-34.431,179.419,5.202,149.075
C05214=1240.400,-125.100,-34.421,179.417,5.203,149.075
C05215=1240.405,-125.350,-34.411,179.415,5.203,149.076
C05216=1240.410,-125.599,-34.402,179.412,5.203,149.077
C05217=1240.415,-125.850,-34.391,179.411,5.203,149.077
C05218=1239.994,-125.860,-34.426,179.406,5.206,149.079
C05219=1239.988,-125.611,-34.436,179.408,5.206,149.079
C05220=1239.983,-125.361,-34.445,179.410,5.206,149.078
C05221=1239.978,-125.110,-34.456,179.413,5.206,149.077
C05222=1239.973,-124.861,-34.466,179.415,5.206,149.077
C05223=1239.968,-124.612,-34.476,179.417,5.206,149.076
C05224=1239.962,-124.362,-34.486,179.419,5.206,149.075
C05225=1239.957,-124.111,-34.496,179.422,5.206,149.075
C05226=1239.952,-123.862,-34.505,179.424,5.206,149.074
C05227=1239.946,-123.613,-34.515,179.426,5.206,149.073
C05228=1239.942,-123.363,-34.525,179.429,5.206,149.073
C05229=1239.937,-123.113,-34.536,179.431,5.206,149.072
C05230=1239.931,-122.863,-34.545,179.434,5.206,149.071
C05231=1239.925,-122.613,-34.555,179.436,5.206,149.070
C05232=1239.921,-122.363,-34.565,179.438,5.206,149.070
C05233=1239.915,-122.114,-34.576,179.441,5.206,149.069
C05234=1239.910,-121.864,-34.586,179.443,5.206,149.068
C05235=1239.905,-121.614,-34.596,179.445,5.206,149.068
C05236=1239.900,-121.365,-34.606,179.447,5.206,149.067
C05237=1239.894,-121.115,-34.616,179.450,5.206,149.066
C05238=1239.889,-120.865,-34.625,179.452,5.206,149.066
C05239=1239.884,-120.615,-34.636,179.454,5.206,149.065
C05240=1239.878,-120.366,-34.646,179.456,5.206,149.064
C05241=1239.873,-120.116,-34.656,179.459,5.207,149.063
C05242=1239.869,-119.866,-34.666,179.461,5.206,149.063
C05243=1239.863,-119.617,-34.676,179.464,5.207,149.062
C05244=1239.857,-119.367,-34.686,179.466,5.206,149.061
C05245=1239.853,-119.117,-34.696,179.468,5.206,149.061
C05246=1239.847,-118.868,-34.707,179.471,5.206,149.060
C05247=1239.842,-118.618,-34.717,179.473,5.206,149.059
C05248=1239.837,-118.368,-34.727,179.476,5.206,149.058
C05249=1239.832,-118.119,-34.737,179.478,5.206,149.058
C05250=1239.826,-117.869,-34.747,179.480,5.206,149.057
C05251=1239.821,-117.619,-34.758,179.482,5.206,149.056
C05252=1239.816,-117.369,-34.768,179.485,5.206,149.056
C05253=1239.811,-117.119,-34.779,179.487,5.206,149.055
C05254=1239.806,-116.870,-34.788,179.489,5.206,149.054
C05255=1239.800,-116.620,-34.798,179.492,5.206,149.053
C05256=1239.795,-116.370,-34.809,179.494,5.206,149.053
C05257=1239.790,-116.120,-34.819,179.496,5.207,149.052
C05258=1239.784,-115.871,-34.829,179.498,5.206,149.051
C05259=1239.780,-115.621,-34.839,179.501,5.207,149.051
C05260=1239.774,-115.371,-34.850,179.503,5.206,149.050
C05261=1239.769,-115.121,-34.860,179.505,5.206,149.049
C05262=1239.764,-114.872,-34.870,179.508,5.206,149.049
C05263=1239.758,-114.622,-34.881,179.510,5.206,149.048
C05264=1239.753,-114.372,-34.891,179.513,5.207,149.047
C05265=1239.748,-114.123,-34.901,179.515,5.206,149.046
C05266=1239.743,-113.872,-34.911,179.517,5.207,149.046
C05267=1239.738,-113.623,-34.922,179.520,5.206,149.045
C05268=1239.732,-113.373,-34.932,179.522,5.207,149.044
C05269=1239.727,-113.123,-34.942,179.524,5.206,149.044
C05270=1239.721,-112.874,-34.953,179.526,5.206,149.043
C05271=1239.716,-112.623,-34.963,179.529,5.206,149.042
C05272=1239.712,-112.375,-34.973,179.531,5.206,149.041
C05273=1239.706,-112.125,-34.984,179.534,5.207,149.041
C05274=1239.701,-111.875,-34.994,179.536,5.206,149.040
C05275=1239.696,-111.625,-35.004,179.539,5.207,149.039
C05276=1239.691,-111.375,-35.015,179.541,5.206,149.039
C05277=1239.685,-111.126,-35.025,179.543,5.207,149.038
C05278=1239.680,-110.875,-35.036,179.546,5.206,149.037
C05279=1239.675,-110.626,-35.047,179.548,5.207,149.036
C05280=1239.670,-110.376,-35.057,179.550,5.206,149.036
C05281=1239.664,-110.127,-35.068,179.552,5.206,149.035
C05282=1239.659,-109.877,-35.078,179.555,5.206,149.034
C05283=1239.654,-109.627,-35.088,179.557,5.206,149.034
C05284=1239.649,-109.378,-35.098,179.560,5.207,149.033
C05285=1239.644,-109.128,-35.109,179.562,5.206,149.032
C05286=1239.638,-108.878,-35.119,179.565,5.207,149.031
C05287=1239.633,-108.628,-35.130,179.567,5.206,149.031
C05288=1239.628,-108.379,-35.140,179.569,5.207,149.030
C05289=1239.623,-108.129,-35.151,179.571,5.206,149.029
C05290=1239.618,-107.879,-35.162,179.574,5.206,149.029
C05291=1239.613,-107.629,-35.172,179.576,5.206,149.028
C05292=1239.607,-107.380,-35.182,179.578,5.206,149.027
C05293=1239.602,-107.130,-35.194,179.581,5.207,149.027
C05294=1239.597,-106.880,-35.204,179.583,5.207,149.026
C05295=1239.592,-106.630,-35.215,179.585,5.207,149.025
C05296=1239.586,-106.381,-35.225,179.587,5.207,149.025
C05297=1239.581,-106.131,-35.236,179.590,5.207,149.024
C05298=1239.576,-105.882,-35.246,179.592,5.207,149.023
C05299=1239.571,-105.631,-35.257,179.595,5.207,149.022
C05300=1239.566,-105.382,-35.268,179.597,5.207,149.022
C05301=1239.561,-105.132,-35.278,179.599,5.206,149.021
C05302=1239.555,-104.883,-35.289,179.602,5.207,149.020
C05303=1239.550,-104.633,-35.300,179.604,5.207,149.020
C05304=1239.545,-104.383,-35.310,179.607,5.207,149.019
C05305=1239.540,-104.133,-35.321,179.609,5.207,149.018
C05306=1239.534,-103.884,-35.332,179.611,5.207,149.017
C05307=1239.529,-103.634,-35.342,179.613,5.207,149.017
C05308=1239.524,-103.384,-35.352,179.616,5.207,149.016
C05309=1239.519,-103.135,-35.364,179.618,5.207,149.015
C05310=1239.514,-102.885,-35.374,179.621,5.207,149.015
C05311=1239.508,-102.635,-35.384,179.623,5.207,149.014
C05312=1239.504,-102.385,-35.396,179.625,5.207,149.013
C05313=1239.497,-102.136,-35.406,179.628,5.207,149.012
C05314=1239.493,-101.886,-35.418,179.630,5.207,149.012
C05315=1239.487,-101.636,-35.428,179.632,5.207,149.011
C05316=1239.482,-101.386,-35.439,179.635,5.207,149.010
C05317=1239.477,-101.137,-35.449,179.637,5.207,149.010
C05318=1239.472,-100.887,-35.460,179.639,5.207,149.009
C05319=1239.466,-100.616,-35.472,179.642,5.207,149.008
C05320=1239.461,-100.346,-35.484,179.645,5.207,149.007
C05321=1239.455,-100.074,-35.495,179.647,5.207,149.006
C05322=1239.449,-99.803,-35.507,179.650,5.207,149.006
C05323=1239.444,-99.555,-35.518,179.652,5.207,149.005
C05324=1239.439,-99.304,-35.529,179.654,5.207,149.004
C05325=1239.434,-99.055,-35.540,179.657,5.207,149.004
C05326=1239.429,-98.805,-35.550,179.659,5.207,149.003
C05327=1239.424,-98.555,-35.562,179.662,5.207,149.002
C05328=1239.418,-98.306,-35.572,179.664,5.207,149.001
C05329=1239.414,-98.056,-35.583,179.666,5.207,149.001
C05330=1239.408,-97.806,-35.594,179.668,5.207,149.000
C05331=1239.403,-97.557,-35.605,179.671,5.208,148.999
C05332=1239.398,-97.307,-35.616,179.674,5.207,148.998
C05333=1239.392,-97.058,-35.627,179.676,5.207,148.998
C05334=1239.387,-96.807,-35.637,179.678,5.207,148.997
C05335=1239.382,-96.557,-35.649,179.681,5.207,148.996
C05336=1239.376,-96.308,-35.659,179.683,5.207,148.996
C05337=1239.372,-96.058,-35.671,179.686,5.207,148.995
C05338=1239.367,-95.808,-35.681,179.688,5.207,148.994
C05339=1239.361,-95.559,-35.692,179.690,5.207,148.993
C05340=1239.356,-95.309,-35.703,179.693,5.207,148.993
C05341=1239.351,-95.059,-35.715,179.695,5.207,148.992
C05342=1239.346,-94.810,-35.726,179.698,5.207,148.991
C05343=1239.341,-94.560,-35.736,179.700,5.207,148.991
C05344=1239.336,-94.310,-35.747,179.702,5.207,148.990
C05345=1239.330,-94.060,-35.758,179.704,5.207,148.989
C05346=1239.325,-93.811,-35.770,179.707,5.208,148.988
C05347=1239.320,-93.562,-35.780,179.709,5.207,148.988
C05348=1239.315,-93.312,-35.791,179.712,5.208,148.987
C05349=1239.309,-93.062,-35.803,179.714,5.207,148.986
C05350=1239.305,-92.812,-35.814,179.717,5.208,148.986
C05351=1239.299,-92.562,-35.824,179.719,5.207,148.985
C05352=1239.293,-92.312,-35.836,179.721,5.208,148.984
C05353=1239.289,-92.063,-35.848,179.723,5.208,148.983
C05354=1239.283,-91.813,-35.858,179.726,5.207,148.983
C05355=1239.278,-91.564,-35.869,179.728,5.208,148.982
C05356=1239.273,-91.314,-35.881,179.730,5.207,148.981
C05357=1239.267,-91.064,-35.891,179.733,5.208,148.981
C05358=1239.263,-90.815,-35.902,179.735,5.207,148.980
C05359=1239.257,-90.565,-35.914,179.738,5.208,148.979
C05360=1239.252,-90.315,-35.925,179.740,5.208,148.978
C05361=1239.247,-90.065,-35.936,179.743,5.208,148.978
C05362=1239.242,-89.816,-35.947,179.745,5.208,148.977
C05363=1239.237,-89.566,-35.959,179.747,5.208,148.976
C05364=1239.231,-89.316,-35.969,179.749,5.208,148.976
C05365=1239.227,-89.067,-35.981,179.752,5.208,148.975
C05366=1239.221,-88.817,-35.992,179.754,5.208,148.974
C05367=1239.217,-88.567,-36.004,179.757,5.208,148.973
C05368=1239.211,-88.318,-36.014,179.759,5.208,148.973
C05369=1239.205,-88.068,-36.026,179.762,5.208,148.972
C05370=1239.201,-87.818,-36.037,179.764,5.208,148.971
C05371=1239.195,-87.568,-36.049,179.766,5.209,148.971
C05372=1239.190,-87.319,-36.060,179.768,5.208,148.970
C05373=1239.185,-87.069,-36.070,179.771,5.207,148.969
C05374=1239.180,-86.819,-36.082,179.774,5.208,148.968
C05375=1239.175,-86.569,-36.094,179.776,5.208,148.968
C05376=1239.170,-86.320,-36.105,179.779,5.208,148.967
C05377=1239.164,-86.071,-36.116,179.781,5.208,148.966
C05378=1239.160,-85.821,-36.128,179.783,5.208,148.965
C05379=1239.154,-85.570,-36.139,179.785,5.208,148.965
C05380=1239.149,-85.321,-36.150,179.788,5.208,148.964
C05381=1239.144,-85.072,-36.161,179.790,5.208,148.963
C05382=1239.138,-84.822,-36.173,179.793,5.208,148.963
C05383=1239.134,-84.572,-36.184,179.795,5.208,148.962
C05384=1239.128,-84.322,-36.196,179.798,5.209,148.961
C05385=1239.123,-84.073,-36.207,179.800,5.208,148.960
C05386=1239.118,-83.823,-36.219,179.802,5.209,148.960
C05387=1239.113,-83.573,-36.230,179.804,5.208,148.959
C05388=1239.108,-83.324,-36.241,179.807,5.209,148.958
C05389=1239.102,-83.074,-36.253,179.809,5.208,148.958
C05390=1239.098,-82.824,-36.264,179.812,5.209,148.957
C05391=1239.092,-82.575,-36.276,179.814,5.209,148.956
C05392=1239.087,-82.325,-36.287,179.817,5.209,148.955
C05393=1239.082,-82.075,-36.299,179.819,5.209,148.955
C05394=1239.077,-81.826,-36.310,179.821,5.209,148.954
C05395=1239.071,-81.576,-36.322,179.823,5.209,148.953
C05396=1239.066,-81.327,-36.333,179.826,5.209,148.953
C05397=1239.061,-81.077,-36.345,179.829,5.209,148.952
C05398=1239.056,-80.827,-36.356,179.831,5.209,148.951
C05399=1239.051,-80.577,-36.368,179.834,5.209,148.950
C05400=1239.046,-80.328,-36.379,179.836,5.208,148.950
C05401=1239.041,-80.078,-36.391,179.838,5.209,148.949
C05402=1239.036,-79.828,-36.402,179.840,5.208,148.948
C05403=1239.030,-79.579,-36.414,179.843,5.209,148.947
C05404=1239.025,-79.329,-36.425,179.845,5.209,148.947
C05405=1239.020,-79.079,-36.437,179.848,5.209,148.946
C05406=1239.015,-78.830,-36.448,179.850,5.209,148.945
C05407=1239.010,-78.580,-36.460,179.853,5.209,148.945
C05408=1239.005,-78.330,-36.472,179.855,5.209,148.944
C05409=1238.999,-78.080,-36.483,179.857,5.209,148.943
C05410=1238.993,-77.831,-36.495,179.859,5.209,148.942
C05411=1238.989,-77.581,-36.506,179.862,5.209,148.942
C05412=1238.983,-77.331,-36.518,179.864,5.209,148.941
C05413=1238.979,-77.082,-36.529,179.867,5.210,148.940
C05414=1238.973,-76.832,-36.541,179.869,5.209,148.940
C05415=1238.969,-76.583,-36.553,179.872,5.210,148.939
C05416=1238.963,-76.333,-36.565,179.874,5.209,148.938
C05417=1238.958,-76.083,-36.577,179.877,5.210,148.937
C05418=1238.953,-75.833,-36.588,179.879,5.209,148.937
C05419=1238.947,-75.584,-36.600,179.882,5.210,148.936
C05420=1238.942,-75.334,-36.611,179.884,5.209,148.935
C05421=1238.937,-75.084,-36.623,179.886,5.210,148.934
C05422=1238.932,-74.835,-36.635,179.888,5.209,148.934
C05423=1238.926,-74.564,-36.648,179.891,5.210,148.933
C05424=1238.920,-74.295,-36.661,179.894,5.210,148.932
C05425=1238.915,-74.024,-36.673,179.896,5.210,148.931
C05426=1238.910,-73.754,-36.686,179.899,5.210,148.931
C05427=1238.905,-73.504,-36.698,179.901,5.210,148.930
C05428=1238.900,-73.254,-36.710,179.904,5.210,148.929
C05429=1238.894,-73.004,-36.722,179.906,5.210,148.929
C05430=1238.890,-72.755,-36.734,179.909,5.210,148.928
C05431=1238.884,-72.506,-36.745,179.911,5.210,148.927
C05432=1238.878,-72.256,-36.757,179.913,5.211,148.926
C05433=1238.874,-72.007,-36.768,179.916,5.210,148.925
C05434=1238.868,-71.757,-36.780,179.919,5.210,148.925
C05435=1238.863,-71.507,-36.793,179.921,5.210,148.924
C05436=1238.858,-71.258,-36.804,179.923,5.210,148.923
C05437=1238.853,-71.008,-36.816,179.925,5.210,148.923
C05438=1238.848,-70.758,-36.828,179.928,5.211,148.922
C05439=1238.842,-70.508,-36.840,179.930,5.210,148.921
C05440=1238.838,-70.259,-36.852,179.933,5.211,148.921
C05441=1238.832,-70.009,-36.864,179.935,5.210,148.920
C05442=1238.827,-69.759,-36.875,179.938,5.211,148.919
C05443=1238.822,-69.510,-36.888,179.940,5.211,148.918
C05444=1238.817,-69.260,-36.899,179.942,5.211,148.918
C05445=1238.812,-69.010,-36.911,179.945,5.211,148.917
C05446=1238.807,-68.761,-36.924,179.947,5.211,148.916
C05447=1238.802,-68.511,-36.935,179.949,5.211,148.916
C05448=1238.796,-68.261,-36.947,179.952,5.211,148.915
C05449=1238.791,-68.012,-36.960,179.955,5.211,148.914
C05450=1238.786,-67.762,-36.971,179.957,5.211,148.913
C05451=1238.780,-67.512,-36.983,179.959,5.211,148.912
C05452=1238.776,-67.263,-36.995,179.962,5.211,148.912
C05453=1238.771,-67.013,-37.007,179.964,5.211,148.911
C05454=1238.765,-66.763,-37.019,179.967,5.211,148.910
C05455=1238.760,-66.514,-37.032,179.969,5.211,148.910
C05456=1238.755,-66.264,-37.043,179.971,5.212,148.909
C05457=1238.750,-66.015,-37.056,179.974,5.211,148.908
C05458=1238.745,-65.765,-37.067,179.976,5.212,148.908
C05459=1238.739,-65.515,-37.079,179.978,5.211,148.907
C05460=1238.734,-65.266,-37.092,179.981,5.212,148.906
C05461=1238.730,-65.016,-37.103,179.983,5.212,148.905
C05462=1238.724,-64.767,-37.116,179.986,5.212,148.905
C05463=1238.720,-64.516,-37.128,179.989,5.212,148.904
C05464=1238.715,-64.267,-37.141,179.991,5.212,148.903
C05465=1238.709,-64.017,-37.153,179.994,5.212,148.902
C05466=1238.704,-63.767,-37.164,179.996,5.212,148.902
C05467=1238.699,-63.518,-37.176,179.998,5.212,148.901
C05468=1238.694,-63.268,-37.188,-179.999,5.212,148.900
C05469=1238.689,-63.019,-37.201,-179.997,5.213,148.900
C05470=1238.683,-62.769,-37.213,-179.995,5.212,148.899
C05471=1238.678,-62.519,-37.225,-179.992,5.213,148.898
C05472=1238.673,-62.269,-37.237,-179.990,5.212,148.897
C05473=1238.668,-62.020,-37.250,-179.987,5.213,148.897
C05474=1238.662,-61.770,-37.262,-179.985,5.213,148.896
C05475=1238.658,-61.520,-37.274,-179.983,5.213,148.895
C05476=1238.653,-61.271,-37.286,-179.980,5.213,148.895
C05477=1238.648,-61.021,-37.299,-179.977,5.213,148.894
C05478=1238.643,-60.772,-37.311,-179.975,5.213,148.893
C05479=1238.637,-60.522,-37.323,-179.973,5.213,148.892
C05480=1238.632,-60.273,-37.336,-179.970,5.213,148.892
C05481=1238.627,-60.023,-37.348,-179.968,5.213,148.891
